legal notes
=================
| SPDX-FileCopyrightText: © 2022 ekvip automation GmbH <info@ekvip.de>
| SPDX-License-Identifier: Apache-2.0
| For details check: Apache-2.0_

.. _Apache-2.0: https://www.apache.org/licenses/LICENSE-2.0

.. </legal notes>

parameters
=================

*)

METHOD win1252IsEqualTo
VAR_INPUT
	(* current string to check *)
	stringToCheck	:POINTER TO BYTE;
	(* ``stringToCheck`` must be equal to expected *)
	expected		:POINTER TO BYTE;
	(* ``TRUE`` means ignore cases; ``FALSE`` means cases must be equal too *)
	ignoreCases		:BOOL;
	(* message if the assertion is false *)
	message			:AssertMessage;
END_VAR
VAR
	(* length of current string to check *)
	lenghtStringToCheck		:UDINT;
	(* length of ``expected`` *)
	lengthExpectedString	:UDINT;
	(* string address we use to compare, if it's case sensitive it's equal to ``stringToCheck`` *)
	usedStringToCheck		:POINTER TO BYTE;
	(* seacrch string address we use to compare, if it's case sensitive it's equal to ``expected`` *)
	usedExpectedString		:POINTER TO BYTE;
END_VAR
VAR CONSTANT
	(* length of an empty string to avoid Tc2_System.MEMCMP with length 0 *)
	EMPTY_STRING_LENGTH		:UDINT := 0;
END_VAR
lenghtStringToCheck := THIS^.getWin1252StringLength(stringToCheck);
lengthExpectedString := THIS^.getWin1252StringLength(expected);

IF (lenghtStringToCheck <> lengthExpectedString) THEN
	THIS^.assertionWasWrong(message, THIS^.getDebugInfo('win1252IsEqualTo'));
	RETURN;
ELSIF (lengthExpectedString = EMPTY_STRING_LENGTH) THEN
	RETURN;
END_IF

usedStringToCheck := THIS^.getNewWin1252UpperCaseString(stringToCheck, lenghtStringToCheck, ignoreCases);
usedExpectedString := THIS^.getNewWin1252UpperCaseString(expected, lengthExpectedString, ignoreCases);

IF (Tc2_System.MEMCMP(
		usedStringToCheck,
		usedExpectedString, 
		lengthExpectedString
	) <> CNM_ReturnTypes.ComparationResult.EQUAL
) THEN
	THIS^.assertionWasWrong(message, THIS^.getDebugInfo('win1252IsEqualTo'));
END_IF;

THIS^.win1252FreeMemory(usedStringToCheck, ignoreCases);
THIS^.win1252FreeMemory(usedExpectedString, ignoreCases);
END_METHOD

(*

short summary
=================
This assertion method for windows-1252 strings checks if the current string ``stringToCheck`` is not equal to the ``unexpected`` string

.. attention:: 
	All strings are handled as null terminated byte streams.
	For windows-1252 is end of the string 16#00

.. <legal notes>

legal notes
=================
| SPDX-FileCopyrightText: © 2022 ekvip automation GmbH <info@ekvip.de>
| SPDX-License-Identifier: Apache-2.0
| For details check: Apache-2.0_

.. _Apache-2.0: https://www.apache.org/licenses/LICENSE-2.0

.. </legal notes>

parameters
=================

*)

METHOD win1252IsNotEqualTo
VAR_INPUT
	(* current string to check *)
	stringToCheck	:POINTER TO BYTE;
	(* ``stringToCheck`` must be not equal to expected *)
	unexpected		:POINTER TO BYTE;
	(* ``TRUE`` means ignore cases; ``FALSE`` means cases must be equal too *)
	ignoreCases		:BOOL;
	(* message if the assertion is false *)
	message			:AssertMessage;
END_VAR
VAR
	(* length of current string to check *)
	lenghtStringToCheck		:UDINT;
	(* length of ``unexpected`` *)
	lengthUnexpectedString	:UDINT;
	(* string address we use to compare, if it's case sensitive it's equal to ``stringToCheck`` *)
	usedStringToCheck		:POINTER TO BYTE;
	(* seacrch string address we use to compare, if it's case sensitive it's equal to ``expected`` *)
	usedUnexpectedString	:POINTER TO BYTE;
END_VAR
VAR CONSTANT
	(* length of an empty string to avoid Tc2_System.MEMCMP with length 0 *)
	EMPTY_STRING_LENGTH		:UDINT := 0;
END_VAR
lenghtStringToCheck := THIS^.getWin1252StringLength(stringToCheck);
lengthUnexpectedString := THIS^.getWin1252StringLength(unexpected);

IF ((lenghtStringToCheck = EMPTY_STRING_LENGTH) AND (lengthUnexpectedString = EMPTY_STRING_LENGTH)) THEN
	THIS^.assertionWasWrong(message, THIS^.getDebugInfo('win1252IsNotEqualTo'));
	RETURN;
END_IF

usedStringToCheck := THIS^.getNewWin1252UpperCaseString(stringToCheck, lenghtStringToCheck, ignoreCases);
usedUnexpectedString := THIS^.getNewWin1252UpperCaseString(unexpected, lengthUnexpectedString, ignoreCases);

IF (Tc2_System.MEMCMP(
		usedStringToCheck,
		usedUnexpectedString, 
		lengthUnexpectedString
	) = CNM_ReturnTypes.ComparationResult.EQUAL
) THEN
	THIS^.assertionWasWrong(message, THIS^.getDebugInfo('win1252IsNotEqualTo'));
END_IF;

THIS^.win1252FreeMemory(usedStringToCheck, ignoreCases);
THIS^.win1252FreeMemory(usedUnexpectedString, ignoreCases);
END_METHOD

(*

short summary
=================
This assertion method checks if the current string ``stringToCheck`` is length
is equal to ``expectedLength``

.. attention:: 
	All strings are handled as null terminated byte streams.
	For windows-1252 is end of the string 16#00

.. <legal notes>

legal notes
=================
| SPDX-FileCopyrightText: © 2022 ekvip automation GmbH <info@ekvip.de>
| SPDX-License-Identifier: Apache-2.0
| For details check: Apache-2.0_

.. _Apache-2.0: https://www.apache.org/licenses/LICENSE-2.0

.. </legal notes>

parameters
=================

*)

METHOD win1252LenghtIsExact
VAR_INPUT
	(* current string to check *)
	stringToCheck	:POINTER TO BYTE;
	(* expected length of ``stringToCheck`` *)
	expectedLength	:UDINT;
	(* message if the assertion is false *)
	message			:AssertMessage;
END_VAR
IF (THIS^.getWin1252StringLength(stringToCheck) <> expectedLength) THEN
	THIS^.assertionWasWrong(message, THIS^.getDebugInfo('win1252LenghtIsExact'));
END_IF
END_METHOD

(*

short summary
=================
This assertion method checks if the current string ``stringToCheck`` is length
is equal or less than to ``maxLength``

.. attention:: 
	All strings are handled as null terminated byte streams.
	For windows-1252 is end of the string 16#00

.. <legal notes>

legal notes
=================
| SPDX-FileCopyrightText: © 2022 ekvip automation GmbH <info@ekvip.de>
| SPDX-License-Identifier: Apache-2.0
| For details check: Apache-2.0_

.. _Apache-2.0: https://www.apache.org/licenses/LICENSE-2.0

.. </legal notes>

parameters
=================

*)

METHOD win1252LenghtIsMax
VAR_INPUT
	(* current string to check *)
	stringToCheck	:POINTER TO BYTE;
	(* upper limit of the length of ``stringToCheck`` *)
	maxLength		:UDINT;
	(* message if the assertion is false *)
	message			:AssertMessage;
END_VAR
IF (THIS^.getWin1252StringLength(stringToCheck) > maxLength) THEN
	THIS^.assertionWasWrong(message, THIS^.getDebugInfo('win1252LenghtIsMax'));
END_IF
END_METHOD

(*

short summary
=================
This assertion method checks if the current string ``stringToCheck`` is length
is equal or grater than to ``minLength``

.. attention:: 
	All strings are handled as null terminated byte streams.
	For windows-1252 is end of the string 16#00

.. <legal notes>

legal notes
=================
| SPDX-FileCopyrightText: © 2022 ekvip automation GmbH <info@ekvip.de>
| SPDX-License-Identifier: Apache-2.0
| For details check: Apache-2.0_

.. _Apache-2.0: https://www.apache.org/licenses/LICENSE-2.0

.. </legal notes>

parameters
=================

*)

METHOD win1252LenghtIsMin
VAR_INPUT
	(* current string to check *)
	stringToCheck	:POINTER TO BYTE;
	(* lower limit of the length of ``stringToCheck`` *)
	minLength		:UDINT;
	(* message if the assertion is false *)
	message			:AssertMessage;
END_VAR
IF (THIS^.getWin1252StringLength(stringToCheck) < minLength) THEN
	THIS^.assertionWasWrong(message, THIS^.getDebugInfo('win1252LenghtIsMin'));
END_IF
END_METHOD

(*

short summary
=================
This assertion method checks if the current string ``stringToCheck`` is length
is equal or grater than ``minLength`` and equal or less than ``maxLength``

.. attention:: 
	All strings are handled as null terminated byte streams.
	For windows-1252 is end of the string 16#00

.. <legal notes>

legal notes
=================
| SPDX-FileCopyrightText: © 2022 ekvip automation GmbH <info@ekvip.de>
| SPDX-License-Identifier: Apache-2.0
| For details check: Apache-2.0_

.. _Apache-2.0: https://www.apache.org/licenses/LICENSE-2.0

.. </legal notes>

parameters
=================

*)

METHOD win1252LengthIsBetween
VAR_INPUT
	(* current string to check *)
	stringToCheck	:POINTER TO BYTE;
	(* lower limit of the string length *)
	minLenght		:UDINT;
	(* upper limit of the string length *)
	maxLenght		:UDINT;
	(* message if the assertion is false *)
	message			:AssertMessage;
END_VAR
VAR
	(* length of ``stringToCheck`` *)
	lenghtStringToCheck	:UDINT;
END_VAR
IF (minLenght > maxLenght) THEN
	THIS^.assertionWasWrong(message, THIS^.getDebugInfo('win1252LengthIsBetween'));
	RETURN;
END_IF

lenghtStringToCheck := THIS^.getWin1252StringLength(stringToCheck);

IF (
	(lenghtStringToCheck < minLenght)
	OR (lenghtStringToCheck > maxLenght)
) THEN
	THIS^.assertionWasWrong(message, THIS^.getDebugInfo('win1252LengthIsBetween'));
END_IF;
END_METHOD

(*

short summary
=================
This assertion method checks if the current string ``stringToCheck`` starts with ``start``

.. attention:: 
	All strings are handled as null terminated byte streams.
	For windows-1252 is end of the string 16#00

.. <legal notes>

legal notes
=================
| SPDX-FileCopyrightText: © 2022 ekvip automation GmbH <info@ekvip.de>
| SPDX-License-Identifier: Apache-2.0
| For details check: Apache-2.0_

.. _Apache-2.0: https://www.apache.org/licenses/LICENSE-2.0

.. </legal notes>

parameters
=================

*)

METHOD win1252StartsWith
VAR_INPUT
	(* current string to check *)
	stringToCheck	:POINTER TO BYTE;
	(* expected start of ``stringToCheck`` *)
	start			:POINTER TO BYTE;
	(* ``TRUE`` means ignore cases; ``FALSE`` means cases must be equal too *)
	ignoreCases		:BOOL;
	(* ``TRUE`` means truncation of spaces on the left side of ``stringToCheck``*)
	trim			:BOOL;
	(* message if the assertion is false *)
	message			:AssertMessage;
END_VAR
VAR
	(* length of current string to check *)
	lenghtStringToCheck	:UDINT;
	(* length of ``start`` *)
	lengthOfStart		:UDINT;
	(* string address we use to compare, if it's case sensitive it's equal to ``stringToCheck`` *)
	usedStringToCheck	:POINTER TO BYTE;
	(* seacrch string address we use to compare, if it's case sensitive it's equal to ``start`` *)
	usedStartString		:POINTER TO BYTE;
END_VAR
lenghtStringToCheck := THIS^.getWin1252StringLength(stringToCheck);
lengthOfStart := THIS^.getWin1252StringLength(start);

THIS^.win1252TrimLeft(stringToCheck, lenghtStringToCheck, trim);

IF (
	NOT THIS^.isContainsCheckNecessary(
		stringToCheck		:= stringToCheck,
		searchString		:= start,
		lenghtStringToCheck	:= lenghtStringToCheck,
		lengthSearchString	:= lengthOfStart,
		additionalText		:= THIS^.getDebugInfo('win1252StartsWith'),
		message				:= message
	)
) THEN
	RETURN;
END_IF

usedStringToCheck := THIS^.getNewWin1252UpperCaseString(stringToCheck, lenghtStringToCheck, ignoreCases);
usedStartString := THIS^.getNewWin1252UpperCaseString(start, lengthOfStart, ignoreCases);

IF (Tc2_System.MEMCMP(
		usedStringToCheck,
		usedStartString, 
		lengthOfStart
	) <> CNM_ReturnTypes.ComparationResult.EQUAL
) THEN
	THIS^.assertionWasWrong(message, THIS^.getDebugInfo('win1252StartsWith'));
END_IF;

THIS^.win1252FreeMemory(usedStringToCheck, ignoreCases);
THIS^.win1252FreeMemory(usedStartString, ignoreCases);
END_METHOD

(*

short summary
=================
This method is used to remove the whitespace from the start of the string.
It does not really remove it, it just moves the start address and decreases
the string length

.. <legal notes>

legal notes
=================
| SPDX-FileCopyrightText: © 2022 ekvip automation GmbH <info@ekvip.de>
| SPDX-License-Identifier: Apache-2.0
| For details check: Apache-2.0_

.. _Apache-2.0: https://www.apache.org/licenses/LICENSE-2.0

.. </legal notes>

parameters
=================

*)

METHOD PROTECTED win1252TrimLeft
VAR_IN_OUT
	(* start address of the string *)
	stringAddress	:POINTER TO BYTE;
	(* length of the string ``stringAddress`` *)
	stringLength	:UDINT;
END_VAR
VAR_INPUT
	(* ``TRUE`` means remove the whitespace, ``FALSE`` means do not remove the whitespace *)
	trimString		:BOOL;
END_VAR
VAR
	(* index of the current character *)
	character		:UDINT;
	(* counter of the whitspace characters *)
	whitespaceCount	:UDINT := 0;
END_VAR
IF ((stringAddress = 0) OR (stringLength <= 0) OR (NOT trimString)) THEN
	RETURN;
END_IF

FOR character := 0 TO (stringLength-1) BY 1 DO
	IF (THIS^.isCharWin1252WhiteSpace(stringAddress[character])) THEN
		whitespaceCount := whitespaceCount + 1;
	ELSE
		EXIT;
	END_IF
END_FOR

stringAddress := ADR(stringAddress[whitespaceCount]);
stringLength := stringLength - whitespaceCount;
END_METHOD

(*

short summary
=================
This method is used to remove the whitespace from the end of the string.
It does not really remove it, it just decreases the string length.

.. <legal notes>

legal notes
=================
| SPDX-FileCopyrightText: © 2022 ekvip automation GmbH <info@ekvip.de>
| SPDX-License-Identifier: Apache-2.0
| For details check: Apache-2.0_

.. _Apache-2.0: https://www.apache.org/licenses/LICENSE-2.0

.. </legal notes>

parameters
=================

*)

METHOD PROTECTED win1252TrimRight
VAR_INPUT
	(* start address of the string *)
	stringAddress	:POINTER TO BYTE;
END_VAR
VAR_IN_OUT
	(* length of the string ``stringAddress`` *)
	stringLength	:UDINT;
END_VAR
VAR_INPUT
	(* ``TRUE`` means remove the whitespace, ``FALSE`` means do not remove the whitespace *)
	trimString		:BOOL;
END_VAR
VAR
	(* index of the current character *)
	character	:LINT;
END_VAR
IF ((stringAddress = 0) OR (stringLength <= 0) OR (NOT trimString)) THEN
	RETURN;
END_IF

FOR character := (stringLength-1) TO 0 BY -1 DO
	IF (THIS^.isCharWin1252WhiteSpace(stringAddress[character])) THEN
		stringLength := stringLength-1;
	ELSE
		RETURN;
	END_IF
END_FOR
END_METHOD

(*

short summary
=================
This method converts the lowercase letters in an 8 bit windows-1252 string to uppercase letters.

.. attention:: 
	All strings are handled as null terminated byte streams.
	For windows-1252 is end of the string 16#00

.. attention::
	Sharp S ß (16#DF) will not converted

.. <legal notes>

legal notes
=================
| SPDX-FileCopyrightText: © 2022 ekvip automation GmbH <info@ekvip.de>
| SPDX-License-Identifier: Apache-2.0
| For details check: Apache-2.0_

.. _Apache-2.0: https://www.apache.org/licenses/LICENSE-2.0

.. </legal notes>

parameters
=================

*)

METHOD PROTECTED win1252UpperCase
VAR_INPUT
	(* string to ucase *)
	stringAddress		:POINTER TO BYTE;
	(* length of the string *)
	stringLength		:UDINT;
END_VAR
VAR
	(* index of the current character *)
	character			:UDINT := 0;
END_VAR
VAR CONSTANT
	(* NUL: $00 *)
	END_OF_STRING							:BYTE := 16#00;
	(* a *)                             	
	LOWERCASE_A								:BYTE := 16#61;
	(* z *)                             	
	LOWERCASE_Z								:BYTE := 16#7A;
	(* ß *)                             	
	LOWERCASE_SHARP_S						:BYTE := 16#DF;
	(* ÿ *)                             	
	LOWERCASE_Y_WITH_DIAERESIS				:BYTE := 16#FF;
	(* Ÿ *)                             	
	UPPERCASE_Y_WITH_DIAERESIS				:BYTE := 16#9F;
	(* à *)                             	
	LOWERCASE_A_WITH_GRAVE					:BYTE := 16#E0;
	(* ö *)                             	
	LOWERCASE_O_WITH_DIAERESIS				:BYTE := 16#F6;
	(* ø *)                             	
	LOWERCASE_O_WITH_SLASH					:BYTE := 16#F8;
	(* þ *)                             	
	LOWERCASE_THORN							:BYTE := 16#FE;
	(* š *)                             	
	LOWERCASE_S_WITH_CARON					:BYTE := 16#9A;
	(* œ *)                             	
	LOWERCASE_OE							:BYTE := 16#9C;
	(* ž *)                             	
	LOWERCASE_Z_WITH_CARON					:BYTE := 16#9E;
	(* difference between lowercase and uppercase except for š,œ and ž *)
	DIFFERENCE_LOWERCASE_UPPERCASE			:BYTE := 16#20;
	(* for š,œ and ž the difference between lowercase and uppercase *)
	DIFFERENCE_LOWERCASE_UPPERCASE_SPECIAL	:BYTE := 16#10;
	(* increment for the character index *)
	INCREMENT_CHARACTER						:UDINT := 1;
END_VAR
IF (stringAddress = 0) THEN
	RETURN;
END_IF

WHILE ((stringAddress[character] <> END_OF_STRING) AND (character <= stringLength)) DO
	CASE stringAddress[character] OF
	LOWERCASE_A..LOWERCASE_Z,
	LOWERCASE_A_WITH_GRAVE..LOWERCASE_O_WITH_DIAERESIS,
	LOWERCASE_O_WITH_SLASH..LOWERCASE_THORN:
		stringAddress[character] := stringAddress[character] - DIFFERENCE_LOWERCASE_UPPERCASE;
	LOWERCASE_S_WITH_CARON,
	LOWERCASE_OE,
	LOWERCASE_Z_WITH_CARON:
		stringAddress[character] := stringAddress[character] - DIFFERENCE_LOWERCASE_UPPERCASE_SPECIAL;
	LOWERCASE_Y_WITH_DIAERESIS:
		stringAddress[character] := UPPERCASE_Y_WITH_DIAERESIS;
	LOWERCASE_SHARP_S:;//for ß do nothing, because there is no capital letter for it
	ELSE;// do nothing, it's no small letter 
	END_CASE
	character := character + INCREMENT_CHARACTER;
END_WHILE
END_METHOD

END_FUNCTION_BLOCK

// ---- Assertor/Assertions/StringAssertion/classes/AbstarctStringPointerAssertions.TcPOU
(*

short summary
=================
Abstract class provides methods for checking whether, 
based on the string lengths an assert statement with contains or contains not,
makes sense

.. <legal notes>

legal notes
=================
| SPDX-FileCopyrightText: © 2022 ekvip automation GmbH <info@ekvip.de>
| SPDX-License-Identifier: Apache-2.0
| For details check: Apache-2.0_

.. _Apache-2.0: https://www.apache.org/licenses/LICENSE-2.0

.. </legal notes>

methods and properties
=======================

*)

{attribute 'reflection'}
FUNCTION_BLOCK INTERNAL ABSTRACT AbstarctStringPointerAssertions EXTENDS AbstactAssertion 
VAR
END_VAR

(*

short summary
=================
This abstract property returns the class name of the concrete object, 
It's for debugging purpose

.. attention:: 
	For derivations: **It is necessary that this property is overridden by the concrete class**

.. <legal notes>

legal notes
=================
| SPDX-FileCopyrightText: © 2022 ekvip automation GmbH <info@ekvip.de>
| SPDX-License-Identifier: Apache-2.0
| For details check: Apache-2.0_

.. _Apache-2.0: https://www.apache.org/licenses/LICENSE-2.0

.. </legal notes>

*)

PROPERTY ABSTRACT className :CNM_AbstractObject.ClassName
GET
END_GET
END_PROPERTY

(*

short summary
=================
Methods for checking whether, based on the string lengths an assert statement with contains makes sense

.. <legal notes>

legal notes
=================
| SPDX-FileCopyrightText: © 2022 ekvip automation GmbH <info@ekvip.de>
| SPDX-License-Identifier: Apache-2.0
| For details check: Apache-2.0_

.. _Apache-2.0: https://www.apache.org/licenses/LICENSE-2.0

.. </legal notes>

parameters
==================
:return: ``FLASE`` means it's not necessary 
to check the string content, ``TRUE`` means
it's necessary to check the string content
to know if the assertion is true or false

*)

METHOD PROTECTED isContainsCheckNecessary :BOOL
VAR_INPUT
	(* current string to check *)
	stringToCheck	:POINTER TO BYTE;
	(* string must be found in ``stringToCheck`` *)
	searchString		:POINTER TO BYTE;
	(* length of current string to check *)
	lenghtStringToCheck	:UDINT;
	(* length of ``searchString`` *)
	lengthSearchString	:UDINT;
	(* just additional text if assert is false *)	
	additionalText		:Tc2_System.T_MaxString;
	(* message if the assertion is false *)
	message				:AssertMessage;
END_VAR
isContainsCheckNecessary := FALSE;
IF (lengthSearchString > lenghtStringToCheck) THEN
	THIS^.assertionWasWrong(message, additionalText);
	RETURN;
ELSIF ((stringToCheck = 0) XOR (searchString = 0)) THEN
	THIS^.assertionWasWrong(message, additionalText);
	RETURN;
ELSIF ((stringToCheck = 0) AND (searchString = 0)) THEN
	RETURN; //assert is true
ELSIF (lengthSearchString = 0) THEN
	RETURN; //assert is true
ELSIF ((lenghtStringToCheck <= 0) AND (lengthSearchString > 0)) THEN
	THIS^.assertionWasWrong(message, additionalText);
	RETURN;
END_IF
isContainsCheckNecessary := TRUE;
END_METHOD

(*

short summary
=================
Methods for checking whether, based on the string lengths an assert statement with containsNo makes sense

.. <legal notes>

legal notes
=================
| SPDX-FileCopyrightText: © 2022 ekvip automation GmbH <info@ekvip.de>
| SPDX-License-Identifier: Apache-2.0
| For details check: Apache-2.0_

.. _Apache-2.0: https://www.apache.org/licenses/LICENSE-2.0

.. </legal notes>

parameters
==================
:return: ``FLASE`` means it's not necessary 
to check the string content, ``TRUE`` means
it's necessary to check the string content
to know if the assertion is true or false

*)

METHOD PROTECTED isContainsNoCheckNecessary :BOOL
VAR_INPUT
	(* current string to check *)
	stringToCheck		:POINTER TO BYTE;
	(* string must be found in ``stringToCheck`` *)
	searchString		:POINTER TO BYTE;
	(* length of current string to check *)
	lenghtStringToCheck	:UDINT;
	(* length of ``searchString`` *)
	lengthSearchString	:UDINT;
	(* just additional text if assert is false *)	
	additionalText		:Tc2_System.T_MaxString;
	(* message if the assertion is false *)
	message				:AssertMessage;
END_VAR
isContainsNoCheckNecessary := FALSE;
IF (lengthSearchString > lenghtStringToCheck) THEN
	RETURN; //assert is true
ELSIF ((stringToCheck = 0) XOR (searchString = 0)) THEN
	RETURN; //assert is true
ELSIF ((stringToCheck = 0) AND (searchString = 0)) THEN
	THIS^.assertionWasWrong(message, additionalText);
	RETURN;
ELSIF (lengthSearchString = 0) THEN
	THIS^.assertionWasWrong(message, additionalText);
	RETURN;
ELSIF ((lenghtStringToCheck <= 0) AND (lengthSearchString > 0)) THEN
	RETURN; //assert is true
END_IF
isContainsNoCheckNecessary := TRUE;
END_METHOD

END_FUNCTION_BLOCK

// ---- Assertor/Assertions/StringAssertion/StringNew/classes/Windows125xStringAssertions.TcPOU
(*

short summary
=================
This class provides assert statements for Windows-1252 and Windows-1251 strings up to 255 characters length. 
Used encoding is specified in ``Tc2_Utilities.GLOBAL_SBCS_TABLE`` global variable

.. attention:: 
	All strings are handled as null-terminated byte streams

.. <legal notes>

legal notes
=================
| SPDX-FileCopyrightText: © 2024 ekvip automation GmbH <info@ekvip.de>
| SPDX-License-Identifier: Apache-2.0
| For details check: Apache-2.0_

.. _Apache-2.0: https://www.apache.org/licenses/LICENSE-2.0

.. </legal notes>

methods and properties
=======================

*)

{attribute 'reflection'}
FUNCTION_BLOCK INTERNAL Windows125xStringAssertions EXTENDS AbstactAssertion IMPLEMENTS IWindows125xStringAssertions
VAR
	(* class to handle the windows-1252 and windows-1251 string assertions *)  
	assertion	:Windows125xStringPointerAssertions();
END_VAR

(*

short summary
=================
This abstract property returns the class name of the concrete object, 
It's for debugging purpose

.. <legal notes>

legal notes
=================
| SPDX-FileCopyrightText: © 2022 ekvip automation GmbH <info@ekvip.de>
| SPDX-License-Identifier: Apache-2.0
| For details check: Apache-2.0_

.. _Apache-2.0: https://www.apache.org/licenses/LICENSE-2.0

.. </legal notes>

*)

PROPERTY className :CNM_AbstractObject.ClassName
GET
className := 'CNM_AssertionInterfaceLib.Windows125xStringAssertions';
END_GET
END_PROPERTY

(*

short summary
=================
This assertion method checks if the current string ``stringToCheck`` contains the search string ``searchString``.
Processed strings must be in UTF-8 encoding

.. <legal notes>

legal notes
=================
| SPDX-FileCopyrightText: © 2024 ekvip automation GmbH <info@ekvip.de>
| SPDX-License-Identifier: Apache-2.0
| For details check: Apache-2.0_

.. _Apache-2.0: https://www.apache.org/licenses/LICENSE-2.0

.. </legal notes>

parameters
=================

*)

METHOD contains : IWindows125xStringAssertions
VAR_INPUT
	(* current string to check *)
	stringToCheck	:Tc2_System.T_MaxString;
	(* string must be found in ``stringToCheck`` *)
	searchString	:Tc2_System.T_MaxString;
	(* ``TRUE`` means ignore cases; ``FALSE`` means that cases must be equal too *)
	ignoreCases		:BOOL;
	(* message if the assertion is false *)
	message			:AssertMessage;
END_VAR
contains := THIS^;

assertion.contains(
	stringToCheck 	:= ADR(stringToCheck),
	searchSTring 	:= ADR(searchString),
	ignoreCases 	:= ignoreCases,
	message 		:= message
);
END_METHOD

(*

short summary
=================
This assertion method checks if the current string ``stringToCheck`` doesn't contain the search string ``searchString``.
Processed strings must be in UTF-8 encoding

.. <legal notes>

legal notes
=================
| SPDX-FileCopyrightText: © 2024 ekvip automation GmbH <info@ekvip.de>
| SPDX-License-Identifier: Apache-2.0
| For details check: Apache-2.0_

.. _Apache-2.0: https://www.apache.org/licenses/LICENSE-2.0

.. </legal notes>

parameters
=================

*)

METHOD containsNo : IWindows125xStringAssertions
VAR_INPUT
	(* current string to check *)
	stringToCheck	:Tc2_System.T_MaxString;
	(* string that must not be found in ``stringToCheck`` *)
	searchString	:Tc2_System.T_MaxString;
	(* ``TRUE`` means ignore cases; ``FALSE`` means that cases must be equal too *)
	ignoreCases		:BOOL;
	(* message if the assertion is false *)
	message			:AssertMessage;
END_VAR
containsNo := THIS^;

THIS^.assertion.containsNo(
	stringToCheck 	:= ADR(stringToCheck),
	searchSTring 	:= ADR(searchString),
	ignoreCases 	:= ignoreCases,
	message 		:= message
);
END_METHOD

(*

short summary
=================
This assertion method checks if the current string ``stringToCheck`` ends with the string ``end``.
Processed strings must be in UTF-8 encoding

.. <legal notes>

legal notes
=================
| SPDX-FileCopyrightText: © 2024 ekvip automation GmbH <info@ekvip.de>
| SPDX-License-Identifier: Apache-2.0
| For details check: Apache-2.0_

.. _Apache-2.0: https://www.apache.org/licenses/LICENSE-2.0

.. </legal notes>

parameters
=================

*)

METHOD endsWith : IWindows125xStringAssertions
VAR_INPUT
	(* current string to check *)
	stringToCheck	:Tc2_System.T_MaxString;
	(* expected end of ``stringToCheck`` *)
	end				:Tc2_System.T_MaxString;
	(* ``TRUE`` means ignore cases; ``FALSE`` means that cases must be equal too *)
	ignoreCases		:BOOL;
	(* ``TRUE`` means truncation of spaces on the right side of ``stringToCheck``*)
	trimRight		:BOOL;
	(* message if the assertion is false *)
	message			:AssertMessage;
END_VAR
endsWith := THIS^;

assertion.endsWith(
	stringToCheck	:= ADR(stringToCheck),
	end				:= ADR(end),
	ignoreCases		:= ignoreCases,
	trimRight		:= trimRight,
	message			:= message
);
END_METHOD

(*

short summary
=================
This assertion method checks if the current string ``stringToCheck`` is empty.
Processed strings must be in UTF-8 encoding

.. <legal notes>

legal notes
=================
| SPDX-FileCopyrightText: © 2024 ekvip automation GmbH <info@ekvip.de>
| SPDX-License-Identifier: Apache-2.0
| For details check: Apache-2.0_

.. _Apache-2.0: https://www.apache.org/licenses/LICENSE-2.0

.. </legal notes>

parameters
=================

*)

METHOD isEmpty : IWindows125xStringAssertions
VAR_INPUT
	(* current string to check *)
	stringToCheck	:Tc2_System.T_MaxString;
	(* message if the assertion is false *)
	message			:AssertMessage;
END_VAR
isEmpty := THIS^;

IF (stringToCheck <> '') THEN
	THIS^.assertionWasWrong(message, THIS^.getDebugInfo('isEmpty'));
END_IF
END_METHOD

(*

short summary
=================
This assertion method checks if the current string ``stringToCheck`` is equal to ``expected``.
Processed strings must be in UTF-8 encoding

.. <legal notes>

legal notes
=================
| SPDX-FileCopyrightText: © 2024 ekvip automation GmbH <info@ekvip.de>
| SPDX-License-Identifier: Apache-2.0
| For details check: Apache-2.0_

.. _Apache-2.0: https://www.apache.org/licenses/LICENSE-2.0

.. </legal notes>

parameters
=================

*)

METHOD isEqualTo : IWindows125xStringAssertions
VAR_INPUT
	(* current string to check *)
	stringToCheck	:Tc2_System.T_MaxString;
	(* ``stringToCheck`` must be equal to expected *)
	expected		:Tc2_System.T_MaxString;
	(* ``TRUE`` means ignore cases; ``FALSE`` means that cases must be equal too *)
	ignoreCases		:BOOL;
	(* message if the assertion is false *)
	message			:AssertMessage;
END_VAR
isEqualTo := THIS^;

assertion.isEqualTo(
	stringToCheck	:= ADR(stringToCheck),
	expected		:= ADR(expected),
	ignoreCases		:= ignoreCases,
	message			:= message
);
END_METHOD

(*

short summary
=================
This assertion method checks if the current string ``stringToCheck`` is not empty.
Processed strings must be in UTF-8 encoding

.. <legal notes>

legal notes
=================
| SPDX-FileCopyrightText: © 2024 ekvip automation GmbH <info@ekvip.de>
| SPDX-License-Identifier: Apache-2.0
| For details check: Apache-2.0_

.. _Apache-2.0: https://www.apache.org/licenses/LICENSE-2.0

.. </legal notes>

parameters
=================

*)

METHOD isNotEmpty : IWindows125xStringAssertions
VAR_INPUT
	(* current string to check *)
	stringToCheck	:Tc2_System.T_MaxString;
	(* message if the assertion is false *)
	message			:AssertMessage;
END_VAR
isNotEmpty := THIS^;

IF (stringToCheck = '') THEN
	THIS^.assertionWasWrong(message, THIS^.getDebugInfo('isEmpty'));
END_IF
END_METHOD

(*

short summary
=================
This assertion method checks if the current string ``stringToCheck`` is not equal to ``unexpected``.
Processed strings must be in UTF-8 encoding

.. <legal notes>

legal notes
=================
| SPDX-FileCopyrightText: © 2024 ekvip automation GmbH <info@ekvip.de>
| SPDX-License-Identifier: Apache-2.0
| For details check: Apache-2.0_

.. _Apache-2.0: https://www.apache.org/licenses/LICENSE-2.0

.. </legal notes>

parameters
=================

*)

METHOD isNotEqualTo : IWindows125xStringAssertions
VAR_INPUT
	(* current string to check *)
	stringToCheck	:Tc2_System.T_MaxString;
	(* ``stringToCheck`` must be not equal to expected *)
	unexpected		:Tc2_System.T_MaxString;
	(* ``TRUE`` means ignore cases; ``FALSE`` means that cases must be equal too *)
	ignoreCases		:BOOL;
	(* message if the assertion is false *)
	message			:AssertMessage;
END_VAR
isNotEqualTo := THIS^;

THIS^.assertion.isNotEqualTo(
	stringToCheck	:= ADR(stringToCheck),
	unexpected		:= ADR(unexpected),
	ignoreCases		:= ignoreCases,
	message			:= message
);
END_METHOD

(*

short summary
=================
This assertion method checks if the current string ``stringToCheck`` length is between ``minLenght`` and ``maxLenght``.
Processed strings must be in UTF-8 encoding

.. <legal notes>

legal notes
=================
| SPDX-FileCopyrightText: © 2024 ekvip automation GmbH <info@ekvip.de>
| SPDX-License-Identifier: Apache-2.0
| For details check: Apache-2.0_

.. _Apache-2.0: https://www.apache.org/licenses/LICENSE-2.0

.. </legal notes>

parameters
=================

*)

METHOD lenghtIsBetween : IWindows125xStringAssertions
VAR_INPUT
	(* current string to check *)
	stringToCheck	:Tc2_System.T_MaxString;
	(* lower limit of the string length *)
	minLenght		:USINT;
	(* upper limit of the string length *)
	maxLenght		:USINT;
	(* message if the assertion is false *)
	message			:AssertMessage;
END_VAR
lenghtIsBetween := THIS^;

THIS^.assertion.lengthIsBetween(
	stringToCheck	:= ADR(stringToCheck),
	minLenght		:= minLenght,
	maxLenght		:= maxLenght,
	message			:= message
);
END_METHOD

(*

short summary
=================
This assertion method checks if the current string ``stringToCheck`` length is equal to ``expectedLength``.
Processed strings must be in UTF-8 encoding

.. <legal notes>

legal notes
=================
| SPDX-FileCopyrightText: © 2024 ekvip automation GmbH <info@ekvip.de>
| SPDX-License-Identifier: Apache-2.0
| For details check: Apache-2.0_

.. _Apache-2.0: https://www.apache.org/licenses/LICENSE-2.0

.. </legal notes>

parameters
=================

*)

METHOD lenghtIsExact : IWindows125xStringAssertions
VAR_INPUT
	(* current string to check *)
	stringToCheck	:Tc2_System.T_MaxString;
	(* expected length of ``stringToCheck`` *)
	expectedLength	:USINT;
	(* message if the assertion is false *)
	message			:AssertMessage;
END_VAR
lenghtIsExact := THIS^;

THIS^.assertion.lenghtIsExact(
	stringToCheck	:= ADR(stringToCheck),
	expectedLength	:= expectedLength,
	message			:= message
);
END_METHOD

(*

short summary
=================
This assertion method checks if the current string ``stringToCheck`` length is equal or less than to ``maxLength``.
Processed strings must be in UTF-8 encoding

.. <legal notes>

legal notes
=================
| SPDX-FileCopyrightText: © 2024 ekvip automation GmbH <info@ekvip.de>
| SPDX-License-Identifier: Apache-2.0
| For details check: Apache-2.0_

.. _Apache-2.0: https://www.apache.org/licenses/LICENSE-2.0

.. </legal notes>

parameters
=================

*)

METHOD lenghtIsMax : IWindows125xStringAssertions
VAR_INPUT
	(* current string to check *)
	stringToCheck	:Tc2_System.T_MaxString;
	(* upper limit of the length of ``stringToCheck`` *)
	maxLength		:USINT;
	(* message if the assertion is false *)
	message			:AssertMessage;
END_VAR
lenghtIsMax := THIS^;

THIS^.assertion.lenghtIsMax(
	stringToCheck	:= ADR(stringToCheck),
	maxLength		:= maxLength,
	message			:= message
);
END_METHOD

(*

short summary
=================
This assertion method checks if the current string ``stringToCheck`` length is equal or grater than to ``minLength``.
Processed strings must be in UTF-8 encoding

.. <legal notes>

legal notes
=================
| SPDX-FileCopyrightText: © 2024 ekvip automation GmbH <info@ekvip.de>
| SPDX-License-Identifier: Apache-2.0
| For details check: Apache-2.0_

.. _Apache-2.0: https://www.apache.org/licenses/LICENSE-2.0

.. </legal notes>

parameters
=================

*)

METHOD lenghtIsMin : IWindows125xStringAssertions
VAR_INPUT
	(* current string to check *)
	stringToCheck	:Tc2_System.T_MaxString;
	(* lower limit of the length of ``stringToCheck`` *)
	minLength		:USINT;
	(* message if the assertion is false *)
	message			:AssertMessage;
END_VAR
lenghtIsMin := THIS^;

THIS^.assertion.lenghtIsMin(
	stringToCheck	:= ADR(stringToCheck),
	minLength		:= minLength,
	message			:= message
);
END_METHOD

(*

short summary
=================
This methods is the setter for the callback class if an assertion was false

.. <legal notes>

legal notes
=================
| SPDX-FileCopyrightText: © 2024 ekvip automation GmbH <info@ekvip.de>
| SPDX-License-Identifier: Apache-2.0
| For details check: Apache-2.0_

.. _Apache-2.0: https://www.apache.org/licenses/LICENSE-2.0

.. </legal notes>

parameters
=================

*)

METHOD setCallBack
VAR_INPUT
	(* the class that must be informed if an assertion is false *)
	callBack	:IAssertCallback;  
END_VAR
SUPER^.setCallBack(callBack);
THIS^.assertion.setCallBack(callBack);
END_METHOD

(*

short summary
=================
This assertion method checks if the current string ``stringToCheck`` starts with string ``start``.
Processed strings must be in UTF-8 encoding

.. <legal notes>

legal notes
=================
| SPDX-FileCopyrightText: © 2024 ekvip automation GmbH <info@ekvip.de>
| SPDX-License-Identifier: Apache-2.0
| For details check: Apache-2.0_

.. _Apache-2.0: https://www.apache.org/licenses/LICENSE-2.0

.. </legal notes>

parameters
=================

*)

METHOD startsWith : IWindows125xStringAssertions
VAR_INPUT
	(* current string to check *)
	stringToCheck	:Tc2_System.T_MaxString;
	(* expected start of ``stringToCheck`` *)
	start			:Tc2_System.T_MaxString;
	(* ``TRUE`` means ignore cases; ``FALSE`` means that cases must be equal too *)
	ignoreCases		:BOOL;
	(* ``TRUE`` means truncation of spaces on the left side of ``stringToCheck``*)
	trimLeft		:BOOL;
	(* message if the assertion is false *)
	message			:AssertMessage;
END_VAR
startsWith := THIS^;

assertion.startsWith(
	stringToCheck	:= ADR(stringToCheck),
	start			:= ADR(start),
	ignoreCases		:= ignoreCases,
	trimLeft		:= trimLeft,
	message			:= message
);
END_METHOD

END_FUNCTION_BLOCK

// ---- Assertor/Assertions/StringAssertion/StringNew/classes/Windows125xStringPointerAssertions.TcPOU
(*

short summary
=================
This class provides assert statements for Windows-1252 and Windows-1251 strings.
Used encoding is specified in ``Tc2_Utilities.GLOBAL_SBCS_TABLE`` global variable

.. attention:: 
	All strings are handled as null-terminated byte streams

.. <legal notes>

legal notes
=================
| SPDX-FileCopyrightText: © 2024 ekvip automation GmbH <info@ekvip.de>
| SPDX-License-Identifier: Apache-2.0
| For details check: Apache-2.0_

.. _Apache-2.0: https://www.apache.org/licenses/LICENSE-2.0

.. </legal notes>

methods and properties
=======================

*)

{attribute 'reflection'}
FUNCTION_BLOCK INTERNAL Windows125xStringPointerAssertions EXTENDS AbstarctStringPointerAssertions IMPLEMENTS IWindows125xStringPointerAssertions

(*

short summary
=================
This abstract property returns the class name of the concrete object, 
It's for debugging purpose

.. <legal notes>

legal notes
=================
| SPDX-FileCopyrightText: © 2024 ekvip automation GmbH <info@ekvip.de>
| SPDX-License-Identifier: Apache-2.0
| For details check: Apache-2.0_

.. _Apache-2.0: https://www.apache.org/licenses/LICENSE-2.0

.. </legal notes>

*)

PROPERTY className :CNM_AbstractObject.ClassName
GET
className := 'CNM_AssertionInterfaceLib.Windows125xStringPointerAssertions';
END_GET
END_PROPERTY

(*

short summary
=================
This assertion method checks if the current string ``stringToCheck`` contains the search string ``searchString``.
Processed strings must be in Windows-1252 or Windows-1251 encoding

.. attention:: 
	All strings are handled as null-terminated byte streams

.. <legal notes>

legal notes
=================
| SPDX-FileCopyrightText: © 2024 ekvip automation GmbH <info@ekvip.de>
| SPDX-License-Identifier: Apache-2.0
| For details check: Apache-2.0_

.. _Apache-2.0: https://www.apache.org/licenses/LICENSE-2.0

.. </legal notes>

parameters
=================

*)

METHOD contains : IWindows125xStringPointerAssertions
VAR_INPUT
	(* current string to check *)
	stringToCheck	:POINTER TO BYTE;
	(* string must be found in ``stringToCheck`` *)
	searchString	:POINTER TO BYTE;
	(* ``TRUE`` means ignore cases; ``FALSE`` means that cases must be equal too *)
	ignoreCases		:BOOL;
	(* message if the assertion is false *)
	message			:AssertMessage;
END_VAR
VAR
	(* length of current string to check *)
	lenghtStringToCheck	:UDINT;
	(* length of ``searchString`` *)
	lengthSearchString	:UDINT;
	(* string address we use to compare, if it's case sensitive it's equal to ``stringToCheck`` *)
	usedStringToCheck	:POINTER TO BYTE;
	(* seacrch string address we use to compare, if it's case sensitive it's equal to ``searchString`` *)
	usedSearchString	:POINTER TO BYTE;
	(* character index for the comperation *)
	character			:UDINT;
END_VAR
contains := THIS^;

lenghtStringToCheck := THIS^.getStringLength(stringToCheck);
lengthSearchString := THIS^.getStringLength(searchString);

IF (
	NOT THIS^.isContainsCheckNecessary(
		stringToCheck		:= stringToCheck,
		searchString		:= searchString,
		lenghtStringToCheck	:= lenghtStringToCheck,
		lengthSearchString	:= lengthSearchString,
		additionalText		:= THIS^.getDebugInfo('contains'),
		message				:= message
	)
) THEN
	RETURN;
END_IF

usedStringToCheck := THIS^.getNewUpperCaseString(stringToCheck, lenghtStringToCheck, ignoreCases);
usedSearchString := THIS^.getNewUpperCaseString(searchString, lengthSearchString, ignoreCases);

FOR (character := 0) TO (lenghtStringToCheck - lengthSearchString) BY 1 DO
	IF (Tc2_System.MEMCMP(
			ADR(usedStringToCheck[character]),
			usedSearchString, 
			lengthSearchString
		) = CNM_ReturnTypes.ComparationResult.EQUAL
	) THEN
		THIS^.freeMemory(usedStringToCheck, ignoreCases);
		THIS^.freeMemory(usedSearchString, ignoreCases);		
		RETURN; //assert is true
	END_IF; 
END_FOR

THIS^.assertionWasWrong(message, THIS^.getDebugInfo('contains'));
THIS^.freeMemory(usedStringToCheck, ignoreCases);
THIS^.freeMemory(usedSearchString, ignoreCases);
END_METHOD

(*

short summary
=================
This assertion method checks if the current string ``stringToCheck`` doesn't contain the search string ``searchString``.
Processed strings must be in Windows-1252 or Windows-1251 encoding

.. attention:: 
	All strings are handled as null-terminated byte streams

.. <legal notes>

legal notes
=================
| SPDX-FileCopyrightText: © 2024 ekvip automation GmbH <info@ekvip.de>
| SPDX-License-Identifier: Apache-2.0
| For details check: Apache-2.0_

.. _Apache-2.0: https://www.apache.org/licenses/LICENSE-2.0

.. </legal notes>

parameters
=================

*)

METHOD containsNo : IWindows125xStringPointerAssertions
VAR_INPUT
	(* current string to check *)
	stringToCheck	:POINTER TO BYTE;
	(* string must be found in ``stringToCheck`` *)
	searchString	:POINTER TO BYTE;
	(* ``TRUE`` means ignore cases; ``FALSE`` means that cases must be equal too *)
	ignoreCases		:BOOL;
	(* message if the assertion is false *)
	message			:AssertMessage;
END_VAR
VAR
	(* length of current string to check *)
	lenghtStringToCheck	:UDINT;
	(* length of ``searchString`` *)
	lengthSearchString	:UDINT;
	(* string address we use to compare, if it's case sensitive it's equal to ``stringToCheck`` *)
	usedStringToCheck	:POINTER TO BYTE;
	(* seacrch string address we use to compare, if it's case sensitive it's equal to ``searchString`` *)
	usedSearchString	:POINTER TO BYTE;
	(* character index for the comperation *)
	character			:UDINT;
END_VAR
containsNo := THIS^;

lenghtStringToCheck := THIS^.getStringLength(stringToCheck);
lengthSearchString := THIS^.getStringLength(searchString);

IF (
	NOT THIS^.isContainsNoCheckNecessary(
		stringToCheck		:= stringToCheck,
		searchString		:= searchString,
		lenghtStringToCheck	:= lenghtStringToCheck,
		lengthSearchString	:= lengthSearchString,
		additionalText		:= THIS^.getDebugInfo('containsNo'),
		message				:= message
	)
) THEN
	RETURN;
END_IF

usedStringToCheck := THIS^.getNewUpperCaseString(stringToCheck, lenghtStringToCheck, ignoreCases);
usedSearchString := THIS^.getNewUpperCaseString(searchString, lengthSearchString, ignoreCases);

FOR (character := 0) TO (lenghtStringToCheck - lengthSearchString) BY 1 DO
	IF (Tc2_System.MEMCMP(
			ADR(usedStringToCheck[character]),
			usedSearchString, 
			lengthSearchString
		) = CNM_ReturnTypes.ComparationResult.EQUAL
	) THEN
		THIS^.assertionWasWrong(message, THIS^.getDebugInfo('containsNo'));
		THIS^.freeMemory(usedStringToCheck, ignoreCases);
		THIS^.freeMemory(usedSearchString, ignoreCases);		
		RETURN;
	END_IF; 
END_FOR

THIS^.freeMemory(usedStringToCheck, ignoreCases);
THIS^.freeMemory(usedSearchString, ignoreCases);
END_METHOD

(*

short summary
=================
This assertion method checks if the current string ``stringToCheck`` ends with the string ``end``.
Processed strings must be in Windows-1252 or Windows-1251 encoding

.. attention:: 
	All strings are handled as null-terminated byte streams

.. <legal notes>

legal notes
=================
| SPDX-FileCopyrightText: © 2024 ekvip automation GmbH <info@ekvip.de>
| SPDX-License-Identifier: Apache-2.0
| For details check: Apache-2.0_

.. _Apache-2.0: https://www.apache.org/licenses/LICENSE-2.0

.. </legal notes>

parameters
=================

*)

METHOD endsWith : IWindows125xStringPointerAssertions
VAR_INPUT
	(* current string to check *)
	stringToCheck	:POINTER TO BYTE;
	(* string must be the end of ``stringToCheck`` *)
	end				:POINTER TO BYTE;
	(* ``TRUE`` means ignore cases; ``FALSE`` means that cases must be equal too *)
	ignoreCases		:BOOL;
	(* ``TRUE`` means truncation of spaces on the right side of ``stringToCheck``*)
	trimRight		:BOOL;
	(* message if the assertion is false *)
	message			:AssertMessage;
END_VAR
VAR
	(* length of current string to check *)
	lenghtStringToCheck	:UDINT;
	(* length of ``end`` *)
	lengthOfEnd			:UDINT;
	(* string address we use to compare, if it's case sensitive it's equal to ``stringToCheck`` *)
	usedStringToCheck	:POINTER TO BYTE;
	(* seacrch string address we use to compare, if it's case sensitive it's equal to ``end`` *)
	usedEndString		:POINTER TO BYTE;
END_VAR
endsWith := THIS^;

lenghtStringToCheck := THIS^.getStringLength(stringToCheck);
lengthOfEnd := THIS^.getStringLength(end);

THIS^.trimRight(stringToCheck, lenghtStringToCheck, trimRight);

IF (
	NOT THIS^.isContainsCheckNecessary(
		stringToCheck		:= stringToCheck,
		searchString		:= end,
		lenghtStringToCheck	:= lenghtStringToCheck,
		lengthSearchString	:= lengthOfEnd,
		additionalText		:= THIS^.getDebugInfo('endsWith'),
		message				:= message
	)
) THEN
	RETURN;
END_IF

usedStringToCheck := THIS^.getNewUpperCaseString(stringToCheck, lenghtStringToCheck, ignoreCases);
usedEndString := THIS^.getNewUpperCaseString(end, lengthOfEnd, ignoreCases);

IF (Tc2_System.MEMCMP(
		ADR(usedStringToCheck[lenghtStringToCheck - lengthOfEnd]),
		usedEndString, 
		lengthOfEnd
	) <> CNM_ReturnTypes.ComparationResult.EQUAL
) THEN
	THIS^.assertionWasWrong(message, THIS^.getDebugInfo('endsWith'));
END_IF;

THIS^.freeMemory(usedStringToCheck, ignoreCases);
THIS^.freeMemory(usedEndString, ignoreCases);
END_METHOD

(*

short summary
=================
This method is used to free allocated memory if needed

.. <legal notes>

legal notes
=================
| SPDX-FileCopyrightText: © 2024 ekvip automation GmbH <info@ekvip.de>
| SPDX-License-Identifier: Apache-2.0
| For details check: Apache-2.0_

.. _Apache-2.0: https://www.apache.org/licenses/LICENSE-2.0

.. </legal notes>

parameters
=================

*)

METHOD PROTECTED freeMemory
VAR_INPUT
	(* start address of the memory to free *)
	stringAddress	:POINTER TO BYTE;
	(* ``TRUE`` means free the memory, ``FALSE`` means do not free the memory *)
	freeMemory		:BOOL;
END_VAR
IF (freeMemory) THEN
	__DELETE(stringAddress);
END_IF
END_METHOD

(*

short summary
=================
this methods copy a string and returns the start address of new string,
all small letters are capitalized in the new string.

.. <legal notes>

legal notes
=================
| SPDX-FileCopyrightText: © 2024 ekvip automation GmbH <info@ekvip.de>
| SPDX-License-Identifier: Apache-2.0
| For details check: Apache-2.0_

.. _Apache-2.0: https://www.apache.org/licenses/LICENSE-2.0

.. </legal notes>

parameters
=================
:return: start address of a string. 
If ``createNewUpperCaseString`` is ``TRUE`` then it's a new string

*)

METHOD PROTECTED getNewUpperCaseString :POINTER TO BYTE; 
VAR_INPUT
	(* start address of the string to copy and capitalize *)
	stringAddress				:POINTER TO BYTE;
	(* length of the string ``stringAddress`` *)
	stringLength				:UDINT;
	(* 
	``TRUE means meake a copy and capitalize it, 
	``FALSE`` means return just ``stringAddress``
	and do nothing else
	*)
	createNewUpperCaseString	:BOOL;
END_VAR
IF (createNewUpperCaseString) THEN
	getNewUpperCaseString := THIS^.getStringCopy(stringAddress, stringLength);
	THIS^.upperCase(getNewUpperCaseString, stringLength);
ELSE
	getNewUpperCaseString := stringAddress;
END_IF
END_METHOD

(*

short summary
=================
this methods copy a string and returns the start address of new string

.. <legal notes>

legal notes
=================
| SPDX-FileCopyrightText: © 2024 ekvip automation GmbH <info@ekvip.de>
| SPDX-License-Identifier: Apache-2.0
| For details check: Apache-2.0_

.. _Apache-2.0: https://www.apache.org/licenses/LICENSE-2.0

.. </legal notes>

parameters
=================
:return: start address of the string copy

*)

METHOD PROTECTED getStringCopy :POINTER TO BYTE
VAR_INPUT
	(* string to copy *)
	stringAddress		:POINTER TO BYTE;
	(* length of the string *)
	stringLength		:UDINT;
END_VAR
getStringCopy := __NEW(BYTE, stringLength);
IF (getStringCopy <> 0) THEN
	Tc2_System.MEMCPY(
		destAddr := getStringCopy,
		srcAddr := stringAddress,
		n := stringLength
	);
END_IF
END_METHOD

(*

short summary
=================
this methods returns the length of a null-terminated string in bytes

.. attention:: 
	All strings are handled as null-terminated byte streams.

.. <legal notes>

legal notes
=================
| SPDX-FileCopyrightText: © 2024 ekvip automation GmbH <info@ekvip.de>
| SPDX-License-Identifier: Apache-2.0
| For details check: Apache-2.0_

.. _Apache-2.0: https://www.apache.org/licenses/LICENSE-2.0

.. </legal notes>

parameters
=================
:return: length of the string

*)

METHOD PROTECTED getStringLength :UDINT
VAR_INPUT
	(* Start address of the string for which the length is to be determined *)
	stringAddress	:POINTER TO BYTE;
END_VAR
VAR CONSTANT
	(* the end of string marker *)
	END_OF_STRING	:BYTE := 16#00;
END_VAR
IF (stringAddress = 0) THEN
	RETURN;
END_IF

WHILE (stringAddress[getStringLength] <> END_OF_STRING) DO
	getStringLength := getStringLength + 1;
END_WHILE
END_METHOD

(*

short summary
=================
this methods checks if a windows-1252 or a windows-1251 character is a whitespace character

.. <legal notes>

legal notes
=================
| SPDX-FileCopyrightText: © 2024 ekvip automation GmbH <info@ekvip.de>
| SPDX-License-Identifier: Apache-2.0
| For details check: Apache-2.0_

.. _Apache-2.0: https://www.apache.org/licenses/LICENSE-2.0

.. </legal notes>

parameters
=================
:return: ``TRUE`` means ``character`` is whitespace,
``FALSE`` means ``character`` is no whitespace 

*)

METHOD PROTECTED isCharWhiteSpace :BOOL
VAR_INPUT
	(* character to check if it's whitespace *)
	character	:BYTE;
END_VAR
VAR CONSTANT
	SPACE			:BYTE := 16#20;
	HORIZONTAL_TAB	:BYTE := 16#09;
	LINE_FEED		:BYTE := 16#0A;
	VERTICAL_TAB	:BYTE := 16#0B;
	FROM_FEED		:BYTE := 16#0C;
	CARRIAGE_RETURN	:BYTE := 16#0D;
END_VAR
CASE character OF
	HORIZONTAL_TAB .. CARRIAGE_RETURN,
	SPACE:
		isCharWhiteSpace := TRUE;
	ELSE
		isCharWhiteSpace := FALSE;	
END_CASE
END_METHOD

(*

short summary
=================
This assertion method checks if the current string ``stringToCheck`` is equal to ``expected``.
Processed strings must be in Windows-1252 or Windows-1251 encoding

.. attention:: 
	All strings are handled as null-terminated byte streams

.. <legal notes>

legal notes
=================
| SPDX-FileCopyrightText: © 2024 ekvip automation GmbH <info@ekvip.de>
| SPDX-License-Identifier: Apache-2.0
| For details check: Apache-2.0_

.. _Apache-2.0: https://www.apache.org/licenses/LICENSE-2.0

.. </legal notes>

parameters
=================

*)

METHOD isEqualTo : IWindows125xStringPointerAssertions
VAR_INPUT
	(* current string to check *)
	stringToCheck	:POINTER TO BYTE;
	(* ``stringToCheck`` must be equal to expected *)
	expected		:POINTER TO BYTE;
	(* ``TRUE`` means ignore cases; ``FALSE`` means that cases must be equal too *)
	ignoreCases		:BOOL;
	(* message if the assertion is false *)
	message			:AssertMessage;
END_VAR
VAR
	(* length of current string to check *)
	lenghtStringToCheck		:UDINT;
	(* length of ``expected`` *)
	lengthExpectedString	:UDINT;
	(* string address we use to compare, if it's case sensitive it's equal to ``stringToCheck`` *)
	usedStringToCheck		:POINTER TO BYTE;
	(* seacrch string address we use to compare, if it's case sensitive it's equal to ``expected`` *)
	usedExpectedString		:POINTER TO BYTE;
END_VAR
VAR CONSTANT
	(* length of an empty string to avoid Tc2_System.MEMCMP with length 0 *)
	EMPTY_STRING_LENGTH		:UDINT := 0;
END_VAR
isEqualTo := THIS^;

lenghtStringToCheck := THIS^.getStringLength(stringToCheck);
lengthExpectedString := THIS^.getStringLength(expected);

IF lenghtStringToCheck <> lengthExpectedString THEN
	THIS^.assertionWasWrong(message, THIS^.getDebugInfo('isEqualTo'));
	RETURN;
ELSIF (lengthExpectedString = EMPTY_STRING_LENGTH) THEN
	RETURN;
END_IF

usedStringToCheck := THIS^.getNewUpperCaseString(stringToCheck, lenghtStringToCheck, ignoreCases);
usedExpectedString := THIS^.getNewUpperCaseString(expected, lengthExpectedString, ignoreCases);

IF (Tc2_System.MEMCMP(
		usedStringToCheck,
		usedExpectedString, 
		lengthExpectedString
	) <> CNM_ReturnTypes.ComparationResult.EQUAL
) THEN
	THIS^.assertionWasWrong(message, THIS^.getDebugInfo('isEqualTo'));
END_IF;

THIS^.freeMemory(usedStringToCheck, ignoreCases);
THIS^.freeMemory(usedExpectedString, ignoreCases);
END_METHOD

(*

short summary
=================
This assertion method checks if the current string ``stringToCheck`` is not equal to ``unexpected``.
Processed strings must be in Windows-1252 or Windows-1251 encoding

.. attention:: 
	All strings are handled as null-terminated byte streams

.. <legal notes>

legal notes
=================
| SPDX-FileCopyrightText: © 2024 ekvip automation GmbH <info@ekvip.de>
| SPDX-License-Identifier: Apache-2.0
| For details check: Apache-2.0_

.. _Apache-2.0: https://www.apache.org/licenses/LICENSE-2.0

.. </legal notes>

parameters
=================

*)

METHOD isNotEqualTo : IWindows125xStringPointerAssertions
VAR_INPUT
	(* current string to check *)
	stringToCheck	:POINTER TO BYTE;
	(* ``stringToCheck`` must be not equal to expected *)
	unexpected		:POINTER TO BYTE;
	(* ``TRUE`` means ignore cases; ``FALSE`` means that cases must be equal too *)
	ignoreCases		:BOOL;
	(* message if the assertion is false *)
	message			:AssertMessage;
END_VAR
VAR
	(* length of current string to check *)
	lenghtStringToCheck		:UDINT;
	(* length of ``unexpected`` *)
	lengthUnexpectedString	:UDINT;
	(* string address we use to compare, if it's case sensitive it's equal to ``stringToCheck`` *)
	usedStringToCheck		:POINTER TO BYTE;
	(* seacrch string address we use to compare, if it's case sensitive it's equal to ``expected`` *)
	usedUnexpectedString	:POINTER TO BYTE;
END_VAR
VAR CONSTANT
	(* length of an empty string to avoid Tc2_System.MEMCMP with length 0 *)
	EMPTY_STRING_LENGTH		:UDINT := 0;
END_VAR
isNotEqualTo := THIS^;

lenghtStringToCheck := THIS^.getStringLength(stringToCheck);
lengthUnexpectedString := THIS^.getStringLength(unexpected);

IF lenghtStringToCheck = EMPTY_STRING_LENGTH AND_THEN lengthUnexpectedString = EMPTY_STRING_LENGTH THEN
	THIS^.assertionWasWrong(message, THIS^.getDebugInfo('isNotEqualTo'));
	RETURN;
END_IF

usedStringToCheck := THIS^.getNewUpperCaseString(stringToCheck, lenghtStringToCheck, ignoreCases);
usedUnexpectedString := THIS^.getNewUpperCaseString(unexpected, lengthUnexpectedString, ignoreCases);

IF (Tc2_System.MEMCMP(
		usedStringToCheck,
		usedUnexpectedString, 
		lengthUnexpectedString
	) = CNM_ReturnTypes.ComparationResult.EQUAL
) THEN
	THIS^.assertionWasWrong(message, THIS^.getDebugInfo('isNotEqualTo'));
END_IF;

THIS^.freeMemory(usedStringToCheck, ignoreCases);
THIS^.freeMemory(usedUnexpectedString, ignoreCases);
END_METHOD

(*

short summary
=================
This assertion method checks if the current string ``stringToCheck`` length is equal to ``expectedLength``.
Processed strings must be in Windows-1252 or Windows-1251 encoding

.. attention:: 
	All strings are handled as null-terminated byte streams

.. <legal notes>

legal notes
=================
| SPDX-FileCopyrightText: © 2024 ekvip automation GmbH <info@ekvip.de>
| SPDX-License-Identifier: Apache-2.0
| For details check: Apache-2.0_

.. _Apache-2.0: https://www.apache.org/licenses/LICENSE-2.0

.. </legal notes>

parameters
=================

*)

METHOD lenghtIsExact : IWindows125xStringPointerAssertions
VAR_INPUT
	(* current string to check *)
	stringToCheck	:POINTER TO BYTE;
	(* expected length of ``stringToCheck`` *)
	expectedLength	:UDINT;
	(* message if the assertion is false *)
	message			:AssertMessage;
END_VAR
lenghtIsExact := THIS^;

IF (THIS^.getStringLength(stringToCheck) <> expectedLength) THEN
	THIS^.assertionWasWrong(message, THIS^.getDebugInfo('lenghtIsExact'));
END_IF
END_METHOD

(*

short summary
=================
This assertion method checks if the current string ``stringToCheck`` length is equal or less than to ``maxLength``.
Processed strings must be in Windows-1252 or Windows-1251 encoding

.. attention:: 
	All strings are handled as null-terminated byte streams

.. <legal notes>

legal notes
=================
| SPDX-FileCopyrightText: © 2024 ekvip automation GmbH <info@ekvip.de>
| SPDX-License-Identifier: Apache-2.0
| For details check: Apache-2.0_

.. _Apache-2.0: https://www.apache.org/licenses/LICENSE-2.0

.. </legal notes>

parameters
=================

*)

METHOD lenghtIsMax : IWindows125xStringPointerAssertions
VAR_INPUT
	(* current string to check *)
	stringToCheck	:POINTER TO BYTE;
	(* upper limit of the length of ``stringToCheck`` *)
	maxLength		:UDINT;
	(* message if the assertion is false *)
	message			:AssertMessage;
END_VAR
lenghtIsMax := THIS^;

IF (THIS^.getStringLength(stringToCheck) > maxLength) THEN
	THIS^.assertionWasWrong(message, THIS^.getDebugInfo('lenghtIsMax'));
END_IF
END_METHOD

(*

short summary
=================
This assertion method checks if the current string ``stringToCheck`` length is equal or grater than to ``minLength``.
Processed strings must be in Windows-1252 or Windows-1251 encoding

.. attention:: 
	All strings are handled as null-terminated byte streams

.. <legal notes>

legal notes
=================
| SPDX-FileCopyrightText: © 2024 ekvip automation GmbH <info@ekvip.de>
| SPDX-License-Identifier: Apache-2.0
| For details check: Apache-2.0_

.. _Apache-2.0: https://www.apache.org/licenses/LICENSE-2.0

.. </legal notes>

parameters
=================

*)

METHOD lenghtIsMin : IWindows125xStringPointerAssertions
VAR_INPUT
	(* current string to check *)
	stringToCheck	:POINTER TO BYTE;
	(* lower limit of the length of ``stringToCheck`` *)
	minLength		:UDINT;
	(* message if the assertion is false *)
	message			:AssertMessage;
END_VAR
lenghtIsMin := THIS^;

IF (THIS^.getStringLength(stringToCheck) < minLength) THEN
	THIS^.assertionWasWrong(message, THIS^.getDebugInfo('lenghtIsMin'));
END_IF
END_METHOD

(*

short summary
=================
This assertion method checks if the current string ``stringToCheck`` length is between ``minLenght`` and ``maxLenght``.
Processed strings must be in Windows-1252 or Windows-1251 encoding

.. attention:: 
	All strings are handled as null-terminated byte streams

.. <legal notes>

legal notes
=================
| SPDX-FileCopyrightText: © 2024 ekvip automation GmbH <info@ekvip.de>
| SPDX-License-Identifier: Apache-2.0
| For details check: Apache-2.0_

.. _Apache-2.0: https://www.apache.org/licenses/LICENSE-2.0

.. </legal notes>

parameters
=================

*)

METHOD lengthIsBetween : IWindows125xStringPointerAssertions
VAR_INPUT
	(* current string to check *)
	stringToCheck	:POINTER TO BYTE;
	(* lower limit of the string length *)
	minLenght		:UDINT;
	(* upper limit of the string length *)
	maxLenght		:UDINT;
	(* message if the assertion is false *)
	message			:AssertMessage;
END_VAR
VAR
	(* length of ``stringToCheck`` *)
	lenghtStringToCheck	:UDINT;
END_VAR
lengthIsBetween := THIS^;

IF minLenght > maxLenght THEN
	THIS^.assertionWasWrong(message, THIS^.getDebugInfo('lengthIsBetween'));
	RETURN;
END_IF

lenghtStringToCheck := THIS^.getStringLength(stringToCheck);

IF lenghtStringToCheck < minLenght OR_ELSE lenghtStringToCheck > maxLenght THEN
	THIS^.assertionWasWrong(message, THIS^.getDebugInfo('lengthIsBetween'));
END_IF;
END_METHOD

(*

short summary
=================
This assertion method checks if the current string ``stringToCheck`` starts with string ``start``.
Processed strings must be in Windows-1252 or Windows-1251 encoding

.. attention:: 
	All strings are handled as null-terminated byte streams

.. <legal notes>

legal notes
=================
| SPDX-FileCopyrightText: © 2024 ekvip automation GmbH <info@ekvip.de>
| SPDX-License-Identifier: Apache-2.0
| For details check: Apache-2.0_

.. _Apache-2.0: https://www.apache.org/licenses/LICENSE-2.0

.. </legal notes>

parameters
=================

*)

METHOD startsWith : IWindows125xStringPointerAssertions
VAR_INPUT
	(* current string to check *)
	stringToCheck	:POINTER TO BYTE;
	(* expected start of ``stringToCheck`` *)
	start			:POINTER TO BYTE;
	(* ``TRUE`` means ignore cases; ``FALSE`` means that cases must be equal too *)
	ignoreCases		:BOOL;
	(* ``TRUE`` means truncation of spaces on the left side of ``stringToCheck``*)
	trimLeft		:BOOL;
	(* message if the assertion is false *)
	message			:AssertMessage;
END_VAR
VAR
	(* length of current string to check *)
	lenghtStringToCheck	:UDINT;
	(* length of ``start`` *)
	lengthOfStart		:UDINT;
	(* string address we use to compare, if it's case sensitive it's equal to ``stringToCheck`` *)
	usedStringToCheck	:POINTER TO BYTE;
	(* seacrch string address we use to compare, if it's case sensitive it's equal to ``start`` *)
	usedStartString		:POINTER TO BYTE;
END_VAR
startsWith := THIS^;

lenghtStringToCheck := THIS^.getStringLength(stringToCheck);
lengthOfStart := THIS^.getStringLength(start);

THIS^.trimLeft(stringToCheck, lenghtStringToCheck, trimLeft);

IF (
	NOT THIS^.isContainsCheckNecessary(
		stringToCheck		:= stringToCheck,
		searchString		:= start,
		lenghtStringToCheck	:= lenghtStringToCheck,
		lengthSearchString	:= lengthOfStart,
		additionalText		:= THIS^.getDebugInfo('startsWith'),
		message				:= message
	)
) THEN
	RETURN;
END_IF

usedStringToCheck := THIS^.getNewUpperCaseString(stringToCheck, lenghtStringToCheck, ignoreCases);
usedStartString := THIS^.getNewUpperCaseString(start, lengthOfStart, ignoreCases);

IF (Tc2_System.MEMCMP(
		usedStringToCheck,
		usedStartString, 
		lengthOfStart
	) <> CNM_ReturnTypes.ComparationResult.EQUAL
) THEN
	THIS^.assertionWasWrong(message, THIS^.getDebugInfo('startsWith'));
END_IF;

THIS^.freeMemory(usedStringToCheck, ignoreCases);
THIS^.freeMemory(usedStartString, ignoreCases);
END_METHOD

(*

short summary
=================
This method is used to remove the whitespace from the start of the string.
It does not really remove it, it just moves the start address and decreases
the string length

.. <legal notes>

legal notes
=================
| SPDX-FileCopyrightText: © 2024 ekvip automation GmbH <info@ekvip.de>
| SPDX-License-Identifier: Apache-2.0
| For details check: Apache-2.0_

.. _Apache-2.0: https://www.apache.org/licenses/LICENSE-2.0

.. </legal notes>

parameters
=================

*)

METHOD PROTECTED trimLeft
VAR_IN_OUT
	(* start address of the string *)
	stringAddress	:POINTER TO BYTE;
	(* length of the string ``stringAddress`` *)
	stringLength	:UDINT;
END_VAR
VAR_INPUT
	(* ``TRUE`` means remove the whitespace, ``FALSE`` means do not remove the whitespace *)
	trimString		:BOOL;
END_VAR
VAR
	(* index of the current character *)
	character		:UDINT;
	(* counter of the whitspace characters *)
	whitespaceCount	:UDINT;
END_VAR
IF (stringAddress = 0 OR_ELSE stringLength <= 0 OR_ELSE NOT trimString) THEN
	RETURN;
END_IF

FOR character := 0 TO stringLength - 1 DO
	IF (THIS^.isCharWhiteSpace(stringAddress[character])) THEN
		whitespaceCount := whitespaceCount + 1;
	ELSE
		EXIT;
	END_IF
END_FOR

stringAddress := ADR(stringAddress[whitespaceCount]);
stringLength := stringLength - whitespaceCount;
END_METHOD

(*

short summary
=================
This method is used to remove the whitespace from the end of the string.
It does not really remove it, it just decreases the string length.

.. <legal notes>

legal notes
=================
| SPDX-FileCopyrightText: © 2024 ekvip automation GmbH <info@ekvip.de>
| SPDX-License-Identifier: Apache-2.0
| For details check: Apache-2.0_

.. _Apache-2.0: https://www.apache.org/licenses/LICENSE-2.0

.. </legal notes>

parameters
=================

*)

METHOD PROTECTED trimRight
VAR_INPUT
	(* start address of the string *)
	stringAddress	:POINTER TO BYTE;
END_VAR
VAR_IN_OUT
	(* length of the string ``stringAddress`` *)
	stringLength	:UDINT;
END_VAR
VAR_INPUT
	(* ``TRUE`` means remove the whitespace, ``FALSE`` means do not remove the whitespace *)
	trimString		:BOOL;
END_VAR
VAR
	(* index of the current character *)
	character	:LINT;
END_VAR
IF stringAddress = 0 OR_ELSE stringLength <= 0 OR_ELSE NOT trimString THEN
	RETURN;
END_IF

FOR character := (stringLength-1) TO 0 BY -1 DO
	IF (THIS^.isCharWhiteSpace(stringAddress[character])) THEN
		stringLength := stringLength-1;
	ELSE
		RETURN;
	END_IF
END_FOR
END_METHOD

(*

short summary
=================
This method converts the lowercase letters in an 8 bit windows-1252 or windows-1251
string to uppercase letters.

.. attention:: 
	All strings are handled as null-terminated byte streams.

.. <legal notes>

legal notes
=================
| SPDX-FileCopyrightText: © 2024 ekvip automation GmbH <info@ekvip.de>
| SPDX-License-Identifier: Apache-2.0
| For details check: Apache-2.0_

.. _Apache-2.0: https://www.apache.org/licenses/LICENSE-2.0

.. </legal notes>

parameters
=================

*)

METHOD PROTECTED upperCase
VAR_INPUT
	(* string to ucase *)
	stringAddress	:POINTER TO BYTE;
	(* length of the string *)
	stringLength	:UDINT;
END_VAR
IF (stringAddress = 0) THEN
	RETURN;
END_IF

CASE Tc2_Utilities.GLOBAL_SBCS_TABLE OF
	Tc2_Utilities.E_SBCSType.eSBCS_WesternEuropean:
		upperCase1252(stringAddress, stringLength);
		
	Tc2_Utilities.E_SBCSType.eSBCS_CentralEuropean:
		upperCase1251(stringAddress, stringLength);
END_CASE
END_METHOD

(*

short summary
=================
This method converts the lowercase letters in an 8 bit windows-1251
string to uppercase letters.

.. attention:: 
	All strings are handled as null-terminated byte streams.

.. <legal notes>

legal notes
=================
| SPDX-FileCopyrightText: © 2024 ekvip automation GmbH <info@ekvip.de>
| SPDX-License-Identifier: Apache-2.0
| For details check: Apache-2.0_

.. _Apache-2.0: https://www.apache.org/licenses/LICENSE-2.0

.. </legal notes>

parameters
=================

*)

METHOD PROTECTED upperCase1251
VAR_INPUT
	(* string to ucase *)
	stringAddress		:POINTER TO BYTE;
	(* length of the string *)
	stringLength		:UDINT;
END_VAR
VAR
	(* index of the current character *)
	character			:UDINT := 0;
END_VAR
VAR CONSTANT
	(* NUL: $00 *)
	END_OF_STRING							:BYTE := 16#00;
	(* a *)                             	
	LOWERCASE_A								:BYTE := 16#61;
	(* z *)                             	
	LOWERCASE_Z								:BYTE := 16#7A;	
	(* а *)
	LOWERCASE_CYRILLIC_A					:BYTE := 16#E0;
	(* я *)
	LOWERCASE_CYRILLIC_YA					:BYTE := 16#FF;
	
	(* ђ *)
	LOWERCASE_CYRILLIC_DJE					:BYTE := 16#90;
	(* љ *)
	LOWERCASE_CYRILLIC_LJE					:BYTE := 16#9A;
	(* њ *)
	LOWERCASE_CYRILLIC_NJE					:BYTE := 16#9C;	
	(* џ *)
	LOWERCASE_CYRILLIC_DZHE					:BYTE := 16#9F;
	(* ё *)
	LOWERCASE_CYRILLIC_IO					:BYTE := 16#B8;
	(* є *)
	LOWERCASE_CYRILLIC_UKRAINIAN_IE			:BYTE := 16#BA;
	(* ї *)
	LOWERCASE_CYRILLIC_YI					:BYTE := 16#BF;

	(* ў *)
	LOWERCASE_CYRILLIC_SHORT_U				:BYTE := 16#A2;
	(* i *)
	LOWERCASE_CYRILLIC_UKRAINIAN_I			:BYTE := 16#B3;
	(* ѕ *)
	LOWERCASE_CYRILLIC_DZE					:BYTE := 16#BE;
	
	(* ѓ *)
	LOWERCASE_CYRILLIC_GJE					:BYTE := 16#83;
	
	(* ґ *)
	LOWERCASE_CYRILLIC_GHE_WITH_UPTURN		:BYTE := 16#B4;
	
	(* ј *)
	LOWERCASE_CYRILLIC_JE					:BYTE := 16#19;
END_VAR
WHILE stringAddress[character] <> END_OF_STRING AND_THEN character <= stringLength DO
	CASE stringAddress[character] OF
		LOWERCASE_A..LOWERCASE_Z,
		LOWERCASE_CYRILLIC_A..LOWERCASE_CYRILLIC_YA:
			stringAddress[character] := stringAddress[character] - 16#20;
		LOWERCASE_CYRILLIC_DJE,
		LOWERCASE_CYRILLIC_LJE,
		LOWERCASE_CYRILLIC_NJE..LOWERCASE_CYRILLIC_DZHE,
		LOWERCASE_CYRILLIC_IO,
		LOWERCASE_CYRILLIC_UKRAINIAN_IE,
		LOWERCASE_CYRILLIC_YI:
			stringAddress[character] := stringAddress[character] - 16#10;
		LOWERCASE_CYRILLIC_SHORT_U,
		LOWERCASE_CYRILLIC_UKRAINIAN_I,
		LOWERCASE_CYRILLIC_DZE:
			stringAddress[character] := 16#01;
		LOWERCASE_CYRILLIC_GJE:
			stringAddress[character] := 16#02;
		LOWERCASE_CYRILLIC_GHE_WITH_UPTURN:
			stringAddress[character] := 16#0F;
		LOWERCASE_CYRILLIC_JE:
			stringAddress[character] := 16#0F;
	END_CASE
	
	character := character + 1;
END_WHILE
END_METHOD

(*

short summary
=================
This method converts the lowercase letters in an 8 bit windows-1252 
string to uppercase letters.

.. attention:: 
	All strings are handled as null terminated byte streams.

.. <legal notes>

legal notes
=================
| SPDX-FileCopyrightText: © 2024 ekvip automation GmbH <info@ekvip.de>
| SPDX-License-Identifier: Apache-2.0
| For details check: Apache-2.0_

.. _Apache-2.0: https://www.apache.org/licenses/LICENSE-2.0

.. </legal notes>

parameters
=================

*)

METHOD PROTECTED upperCase1252
VAR_INPUT
	(* string to ucase *)
	stringAddress		:POINTER TO BYTE;
	(* length of the string *)
	stringLength		:UDINT;
END_VAR
VAR
	(* index of the current character *)
	character			:UDINT := 0;
END_VAR
VAR CONSTANT
	(* NUL: $00 *)
	END_OF_STRING							:BYTE := 16#00;
	(* a *)                             	
	LOWERCASE_A								:BYTE := 16#61;
	(* z *)                             	
	LOWERCASE_Z								:BYTE := 16#7A;
	(* ß *)                             	
	LOWERCASE_SHARP_S						:BYTE := 16#DF;
	(* ÿ *)                             	
	LOWERCASE_Y_WITH_DIAERESIS				:BYTE := 16#FF;
	(* Ÿ *)                             	
	UPPERCASE_Y_WITH_DIAERESIS				:BYTE := 16#9F;
	(* à *)                             	
	LOWERCASE_A_WITH_GRAVE					:BYTE := 16#E0;
	(* ö *)                             	
	LOWERCASE_O_WITH_DIAERESIS				:BYTE := 16#F6;
	(* ø *)                             	
	LOWERCASE_O_WITH_SLASH					:BYTE := 16#F8;
	(* þ *)                             	
	LOWERCASE_THORN							:BYTE := 16#FE;
	(* š *)                             	
	LOWERCASE_S_WITH_CARON					:BYTE := 16#9A;
	(* œ *)                             	
	LOWERCASE_OE							:BYTE := 16#9C;
	(* ž *)                             	
	LOWERCASE_Z_WITH_CARON					:BYTE := 16#9E;
	(* difference between lowercase and uppercase except for š,œ and ž *)
	DIFFERENCE_LOWERCASE_UPPERCASE			:BYTE := 16#20;
	(* for š,œ and ž the difference between lowercase and uppercase *)
	DIFFERENCE_LOWERCASE_UPPERCASE_SPECIAL	:BYTE := 16#10;
END_VAR
WHILE stringAddress[character] <> END_OF_STRING AND_THEN character <= stringLength DO
	CASE stringAddress[character] OF
		LOWERCASE_A..LOWERCASE_Z,
		LOWERCASE_A_WITH_GRAVE..LOWERCASE_O_WITH_DIAERESIS,
		LOWERCASE_O_WITH_SLASH..LOWERCASE_THORN:
			stringAddress[character] := stringAddress[character] - DIFFERENCE_LOWERCASE_UPPERCASE;
		LOWERCASE_S_WITH_CARON,
		LOWERCASE_OE,
		LOWERCASE_Z_WITH_CARON:
			stringAddress[character] := stringAddress[character] - DIFFERENCE_LOWERCASE_UPPERCASE_SPECIAL;
		LOWERCASE_Y_WITH_DIAERESIS:
			stringAddress[character] := UPPERCASE_Y_WITH_DIAERESIS;
		LOWERCASE_SHARP_S:;//for ß do nothing, because there is no capital letter for it
	END_CASE
	
	character := character + 1;
END_WHILE
END_METHOD

END_FUNCTION_BLOCK

// ---- Assertor/Assertions/StringAssertion/WString/classes/utf16StringAssertions.TcPOU
(*

short summary
=================
This class provides assert statements for UTF-16 strings until 255 ``WORD`` length

.. <legal notes>

legal notes
=================
| SPDX-FileCopyrightText: © 2022 ekvip automation GmbH <info@ekvip.de>
| SPDX-License-Identifier: Apache-2.0
| For details check: Apache-2.0_

.. _Apache-2.0: https://www.apache.org/licenses/LICENSE-2.0

.. </legal notes>

methods and properties
=======================

*)

{attribute 'reflection'}
FUNCTION_BLOCK INTERNAL utf16StringAssertions EXTENDS AbstactAssertion IMPLEMENTS IUtf16StringAssertions
VAR
	(* class to handle the UTF-16 string assertions *)  
	assertion	:Utf16StringPointerAssertions();
END_VAR

(*

short summary
=================
This abstract property returns the class name of the concrete object, 
It's for debugging purpose

.. <legal notes>

legal notes
=================
| SPDX-FileCopyrightText: © 2022 ekvip automation GmbH <info@ekvip.de>
| SPDX-License-Identifier: Apache-2.0
| For details check: Apache-2.0_

.. _Apache-2.0: https://www.apache.org/licenses/LICENSE-2.0

.. </legal notes>

*)

PROPERTY className :CNM_AbstractObject.ClassName
GET
className := 'CNM_AssertionInterfaceLib.utf16StringAssertions';
END_GET
END_PROPERTY

(*

short summary
=================
This assertion method for UTF-16 strings checks if the current string ``stringToCheck`` contains the search string ``searchString``

.. <legal notes>

legal notes
=================
| SPDX-FileCopyrightText: © 2022 ekvip automation GmbH <info@ekvip.de>
| SPDX-License-Identifier: Apache-2.0
| For details check: Apache-2.0_

.. _Apache-2.0: https://www.apache.org/licenses/LICENSE-2.0

.. </legal notes>

parameters
=================

*)

METHOD contains
VAR_INPUT
	(* current string to check *)
	stringToCheck	:WSTRING(Tc2_System.MAX_STRING_LENGTH);
	(* string must be found in ``stringToCheck`` *)
	searchString	:WSTRING(Tc2_System.MAX_STRING_LENGTH);
	(* ``TRUE`` means ignore cases; ``FALSE`` means cases must be equal too *)
	ignoreCases		:BOOL;
	(* message if the assertion is false *)
	message			:AssertMessage;
END_VAR
THIS^.assertion.utf16Contains(
	stringToCheck 	:= ADR(stringToCheck),
	searchSTring 	:= ADR(searchString),
	ignoreCases 	:= ignoreCases,
	message 		:= message
);
END_METHOD

(*

short summary
=================
This assertion method for UTF-16 strings checks if the current string ``stringToCheck`` contains not the search string ``searchString``

.. <legal notes>

legal notes
=================
| SPDX-FileCopyrightText: © 2022 ekvip automation GmbH <info@ekvip.de>
| SPDX-License-Identifier: Apache-2.0
| For details check: Apache-2.0_

.. _Apache-2.0: https://www.apache.org/licenses/LICENSE-2.0

.. </legal notes>

parameters
=================

*)

METHOD containsNo
VAR_INPUT
	(* current string to check *)
	stringToCheck	:WSTRING(Tc2_System.MAX_STRING_LENGTH);
	(* string that must not be found in ``stringToCheck`` *)
	searchString	:WSTRING(Tc2_System.MAX_STRING_LENGTH);
	(* ``TRUE`` means ignore cases; ``FALSE`` means cases must be equal too *)
	ignoreCases		:BOOL;
	(* message if the assertion is false *)
	message			:AssertMessage;
END_VAR
THIS^.assertion.utf16ContainsNo(
	stringToCheck 	:= ADR(stringToCheck),
	searchSTring 	:= ADR(searchString),
	ignoreCases 	:= ignoreCases,
	message 		:= message
);
END_METHOD

(*

short summary
=================
This assertion method for UTF-16 strings checks if the current string ``stringToCheck`` ends with the string ``end``

.. attention:: 
	end of the string is **ALWAYS** the right side of the string 
	even for writings which written from right to left like Hebrew or Arabic

.. <legal notes>

legal notes
=================
| SPDX-FileCopyrightText: © 2022 ekvip automation GmbH <info@ekvip.de>
| SPDX-License-Identifier: Apache-2.0
| For details check: Apache-2.0_

.. _Apache-2.0: https://www.apache.org/licenses/LICENSE-2.0

.. </legal notes>

parameters
=================

*)

METHOD endsWith
VAR_INPUT
	(* current string to check *)
	stringToCheck	:WSTRING(Tc2_System.MAX_STRING_LENGTH);
	(* expected end of ``stringToCheck`` *)
	end				:WSTRING(Tc2_System.MAX_STRING_LENGTH);
	(* ``TRUE`` means ignore cases; ``FALSE`` means cases must be equal too *)
	ignoreCases		:BOOL;
	(* ``TRUE`` means truncation of spaces on the right side of ``stringToCheck``*)
	trim			:BOOL;
	(* message if the assertion is false *)
	message			:AssertMessage;
END_VAR
THIS^.assertion.utf16EndsWith(
	stringToCheck	:= ADR(stringToCheck),
	end				:= ADR(end),
	ignoreCases		:= ignoreCases,
	trim			:= trim,
	message			:= message
);
END_METHOD

(*

short summary
=================
This assertion method checks if the current string ``stringToCheck`` is empty

.. <legal notes>

legal notes
=================
| SPDX-FileCopyrightText: © 2022 ekvip automation GmbH <info@ekvip.de>
| SPDX-License-Identifier: Apache-2.0
| For details check: Apache-2.0_

.. _Apache-2.0: https://www.apache.org/licenses/LICENSE-2.0

.. </legal notes>

parameters
=================

*)

METHOD isEmpty
VAR_INPUT
	(* current string to check *)
	stringToCheck	:WSTRING(Tc2_System.MAX_STRING_LENGTH);
	(* message if the assertion is false *)
	message			:AssertMessage;
END_VAR
IF (stringToCheck <> "") THEN
	THIS^.assertionWasWrong(message, THIS^.getDebugInfo('isEmpty'));
END_IF
END_METHOD

(*

short summary
=================
This assertion method checks if the current string ``stringToCheck`` is equal to ``expected``

.. <legal notes>

legal notes
=================
| SPDX-FileCopyrightText: © 2022 ekvip automation GmbH <info@ekvip.de>
| SPDX-License-Identifier: Apache-2.0
| For details check: Apache-2.0_

.. _Apache-2.0: https://www.apache.org/licenses/LICENSE-2.0

.. </legal notes>

parameters
=================

*)

METHOD isEqualTo
VAR_INPUT
	(* current string to check *)
	stringToCheck	:WSTRING(Tc2_System.MAX_STRING_LENGTH);
	(* ``stringToCheck`` must be equal to expected *)
	expected		:WSTRING(Tc2_System.MAX_STRING_LENGTH);
	(* ``TRUE`` means ignore cases; ``FALSE`` means cases must be equal too *)
	ignoreCases		:BOOL;
	(* message if the assertion is false *)
	message			:AssertMessage;
END_VAR
THIS^.assertion.utf16IsEqualTo(
	stringToCheck	:= ADR(stringToCheck),
	expected		:= ADR(expected),
	ignoreCases		:= ignoreCases,
	message			:= message
);
END_METHOD

(*

short summary
=================
This assertion method checks if the current string ``stringToCheck`` is not empty

.. <legal notes>

legal notes
=================
| SPDX-FileCopyrightText: © 2022 ekvip automation GmbH <info@ekvip.de>
| SPDX-License-Identifier: Apache-2.0
| For details check: Apache-2.0_

.. _Apache-2.0: https://www.apache.org/licenses/LICENSE-2.0

.. </legal notes>

parameters
=================

*)

METHOD isNotEmpty
VAR_INPUT
	(* current string to check *)
	stringToCheck	:WSTRING(Tc2_System.MAX_STRING_LENGTH);
	(* message if the assertion is false *)
	message			:AssertMessage;
END_VAR
IF (stringToCheck = "") THEN
	THIS^.assertionWasWrong(message, THIS^.getDebugInfo('isNotEmpty'));
END_IF
END_METHOD

(*

short summary
=================
This assertion method checks if the current string ``stringToCheck`` is not equal to ``unexpected``

.. <legal notes>

legal notes
=================
| SPDX-FileCopyrightText: © 2022 ekvip automation GmbH <info@ekvip.de>
| SPDX-License-Identifier: Apache-2.0
| For details check: Apache-2.0_

.. _Apache-2.0: https://www.apache.org/licenses/LICENSE-2.0

.. </legal notes>

parameters
=================

*)

METHOD isNotEqualTo
VAR_INPUT
	(* current string to check *)
	stringToCheck	:WSTRING(Tc2_System.MAX_STRING_LENGTH);
	(* ``stringToCheck`` must be not equal to expected *)
	unexpected		:WSTRING(Tc2_System.MAX_STRING_LENGTH);
	(* ``TRUE`` means ignore cases; ``FALSE`` means cases must be equal too *)
	ignoreCases		:BOOL;
	(* message if the assertion is false *)
	message			:AssertMessage;
END_VAR
THIS^.assertion.utf16IsNotEqualTo(
	stringToCheck	:= ADR(stringToCheck),
	unexpected		:= ADR(unexpected),
	ignoreCases		:= ignoreCases,
	message			:= message
);
END_METHOD

(*

short summary
=================
This assertion method checks if the current string ``stringToCheck`` length
is between ``minLenght`` and ``maxLenght``

.. <legal notes>

legal notes
=================
| SPDX-FileCopyrightText: © 2022 ekvip automation GmbH <info@ekvip.de>
| SPDX-License-Identifier: Apache-2.0
| For details check: Apache-2.0_

.. _Apache-2.0: https://www.apache.org/licenses/LICENSE-2.0

.. </legal notes>

parameters
=================

*)

METHOD lenghtIsBetween
VAR_INPUT
	(* current string to check *)
	stringToCheck	:WSTRING(Tc2_System.MAX_STRING_LENGTH);
	(* lower limit of the string length *)
	minLenght		:USINT;
	(* upper limit of the string length *)
	maxLenght		:USINT;
	(* message if the assertion is false *)
	message			:AssertMessage;
END_VAR
THIS^.assertion.utf16LengthIsBetween(
	stringToCheck	:= ADR(stringToCheck),
	minLenght		:= minLenght,
	maxLenght		:= maxLenght,
	message			:= message
);
END_METHOD

(*

short summary
=================
This assertion method checks if the current string ``stringToCheck`` length
is equal to ``expectedLength``

.. <legal notes>

legal notes
=================
| SPDX-FileCopyrightText: © 2022 ekvip automation GmbH <info@ekvip.de>
| SPDX-License-Identifier: Apache-2.0
| For details check: Apache-2.0_

.. _Apache-2.0: https://www.apache.org/licenses/LICENSE-2.0

.. </legal notes>

parameters
=================

*)

METHOD lenghtIsExact
VAR_INPUT
	(* current string to check *)
	stringToCheck	:WSTRING(Tc2_System.MAX_STRING_LENGTH);
	(* expected length of ``stringToCheck`` *)
	expectedLength	:USINT;
	(* message if the assertion is false *)
	message			:AssertMessage;
END_VAR
THIS^.assertion.utf16LenghtIsExact(
	stringToCheck	:= ADR(stringToCheck),
	expectedLength	:= expectedLength,
	message			:= message
);
END_METHOD

(*

short summary
=================
This assertion method checks if the current string ``stringToCheck`` length
is equal or less than to ``maxLength``

.. <legal notes>

legal notes
=================
| SPDX-FileCopyrightText: © 2022 ekvip automation GmbH <info@ekvip.de>
| SPDX-License-Identifier: Apache-2.0
| For details check: Apache-2.0_

.. _Apache-2.0: https://www.apache.org/licenses/LICENSE-2.0

.. </legal notes>

parameters
=================

*)

METHOD lenghtIsMax
VAR_INPUT
	(* current string to check *)
	stringToCheck	:WSTRING(Tc2_System.MAX_STRING_LENGTH);
	(* upper limit of the length of ``stringToCheck`` *)
	maxLength		:USINT;
	(* message if the assertion is false *)
	message			:AssertMessage;
END_VAR
THIS^.assertion.utf16LenghtIsMax(
	stringToCheck	:= ADR(stringToCheck),
	maxLength		:= maxLength,
	message			:= message
);
END_METHOD

(*

short summary
=================
This assertion method checks if the current string ``stringToCheck`` length
is equal or grater than to ``minLength``

.. <legal notes>

legal notes
=================
| SPDX-FileCopyrightText: © 2022 ekvip automation GmbH <info@ekvip.de>
| SPDX-License-Identifier: Apache-2.0
| For details check: Apache-2.0_

.. _Apache-2.0: https://www.apache.org/licenses/LICENSE-2.0

.. </legal notes>

parameters
=================

*)

METHOD lenghtIsMin
VAR_INPUT
	(* current string to check *)
	stringToCheck	:WSTRING(Tc2_System.MAX_STRING_LENGTH);
	(* lower limit of the length of ``stringToCheck`` *)
	minLength		:USINT;
	(* message if the assertion is false *)
	message			:AssertMessage;
END_VAR
THIS^.assertion.utf16LenghtIsMin(
	stringToCheck	:= ADR(stringToCheck),
	minLength		:= minLength,
	message			:= message
);
END_METHOD

(*

short summary
=================
This methods is the setter for the callback class if an assertion was false

.. <legal notes>

legal notes
=================
| SPDX-FileCopyrightText: © 2022 ekvip automation GmbH <info@ekvip.de>
| SPDX-License-Identifier: Apache-2.0
| For details check: Apache-2.0_

.. _Apache-2.0: https://www.apache.org/licenses/LICENSE-2.0

.. </legal notes>

parameters
=================

*)

METHOD setCallBack
VAR_INPUT
	(* the class that must be informed if an assertion is false *)
	callBack	:IAssertCallback;  
END_VAR
SUPER^.setCallBack(callBack);
THIS^.assertion.setCallBack(callBack);
END_METHOD

(*

short summary
=================
This assertion method checks if the current string ``stringToCheck`` starts with ``start``

.. attention:: 
	start of the string is **ALWAYS** the left side of the string 
	even for writings which written from right to left like Hebrew or Arabic

.. <legal notes>

legal notes
=================
| SPDX-FileCopyrightText: © 2022 ekvip automation GmbH <info@ekvip.de>
| SPDX-License-Identifier: Apache-2.0
| For details check: Apache-2.0_

.. _Apache-2.0: https://www.apache.org/licenses/LICENSE-2.0

.. </legal notes>

parameters
=================

*)

METHOD startsWith
VAR_INPUT
	(* current string to check *)
	stringToCheck	:WSTRING(Tc2_System.MAX_STRING_LENGTH);
	(* expected start of ``stringToCheck`` *)
	start			:WSTRING(Tc2_System.MAX_STRING_LENGTH);
	(* ``TRUE`` means ignore cases; ``FALSE`` means cases must be equal too *)
	ignoreCases		:BOOL;
	(* ``TRUE`` means truncation of spaces on the left side of ``stringToCheck``*)
	trim			:BOOL;
	(* message if the assertion is false *)
	message			:AssertMessage;
END_VAR
THIS^.assertion.utf16StartsWith(
	stringToCheck	:= ADR(stringToCheck),
	start			:= ADR(start),
	ignoreCases		:= ignoreCases,
	trim			:= trim,
	message			:= message
);
END_METHOD

END_FUNCTION_BLOCK

// ---- Assertor/Assertions/StringAssertion/WString/classes/Utf16StringPointerAssertions.TcPOU
(*

short summary
=================
This class provides assert statements for UTF-16 strings

.. attention:: 
	All strings are handled as null terminated word streams.
	For UTF-16 is end of the string 16#00_00

.. <legal notes>

legal notes
=================
| SPDX-FileCopyrightText: © 2022 ekvip automation GmbH <info@ekvip.de>
| SPDX-License-Identifier: Apache-2.0
| For details check: Apache-2.0_

.. _Apache-2.0: https://www.apache.org/licenses/LICENSE-2.0

.. </legal notes>

methods and properties
=======================

*)

{attribute 'reflection'}
FUNCTION_BLOCK INTERNAL Utf16StringPointerAssertions EXTENDS AbstarctStringPointerAssertions IMPLEMENTS IUtf16StringPointerAssertions
VAR
END_VAR

(*

short summary
=================
This abstract property returns the class name of the concrete object, 
It's for debugging purpose

.. <legal notes>

legal notes
=================
| SPDX-FileCopyrightText: © 2022 ekvip automation GmbH <info@ekvip.de>
| SPDX-License-Identifier: Apache-2.0
| For details check: Apache-2.0_

.. _Apache-2.0: https://www.apache.org/licenses/LICENSE-2.0

.. </legal notes>

*)

PROPERTY className :CNM_AbstractObject.ClassName
GET
className := 'CNM_AssertionInterfaceLib.Utf16StringPointerAssertions';
END_GET
END_PROPERTY

(*

short summary
=================
this methods copy a string and returns the start address of new string

.. <legal notes>

legal notes
=================
| SPDX-FileCopyrightText: © 2022 ekvip automation GmbH <info@ekvip.de>
| SPDX-License-Identifier: Apache-2.0
| For details check: Apache-2.0_

.. _Apache-2.0: https://www.apache.org/licenses/LICENSE-2.0

.. </legal notes>

parameters
=================
:return: start address of the UTF-16 string copy

*)

METHOD PROTECTED getCopyOfUtf16String :POINTER TO WORD
VAR_INPUT
	(* string to copy *)
	stringAddress		:POINTER TO WORD;
	(* length of the string in words*)
	stringLengthInWord	:UDINT;
END_VAR
getCopyOfUtf16String := __NEW(WORD, stringLengthInWord);
IF (getCopyOfUtf16String <> 0) THEN
	Tc2_System.MEMCPY(
		destAddr := getCopyOfUtf16String,
		srcAddr := stringAddress,
		n := stringLengthInWord * SIZEOF(WORD)
	);
END_IF
END_METHOD

(*

short summary
=================
this methods copy a string and returns the start address of new string,
all small letters are capitalized in the new string.

.. <legal notes>

legal notes
=================
| SPDX-FileCopyrightText: © 2022 ekvip automation GmbH <info@ekvip.de>
| SPDX-License-Identifier: Apache-2.0
| For details check: Apache-2.0_

.. _Apache-2.0: https://www.apache.org/licenses/LICENSE-2.0

.. </legal notes>

parameters
=================
:return: start address of the UTF-16 string. 
If ``createNewUpperCaseString`` is ``TRUE`` then it's a new string

*)

METHOD PROTECTED getNewUtf16UCaseString :POINTER TO WORD; 
VAR_INPUT
	(* start address of the string to copy and capitalize *)
	stringAddress				:POINTER TO WORD;
	(* length of the string ``stringAddress`` *)
	stringLengthInWord			:UDINT;
	(* 
	``TRUE means meake a copy and capitalize it, 
	``FALSE`` means return just ``stringAddress``
	and do nothing else
	*)
	createNewUpperCaseString	:BOOL;
END_VAR
IF (createNewUpperCaseString) THEN
	getNewUtf16UCaseString := THIS^.getCopyOfUtf16String(stringAddress, stringLengthInWord);
	THIS^.utf16UpperCase(getNewUtf16UCaseString, stringLengthInWord);
ELSE
	getNewUtf16UCaseString := stringAddress;
END_IF
END_METHOD

(*

short summary
=================
This methods returns the length of a null terminated UTF-16 string.
The returned length is in characters (in UTF-16 have some charcters 32 bit length).
This method provides two outputs to get the length in byte and word, too. 

.. attention:: 
	All strings are handled as null terminated byte streams.
	For UTF-16 is end of the string 16#00_00

.. <legal notes>

legal notes
=================
| SPDX-FileCopyrightText: © 2022 ekvip automation GmbH <info@ekvip.de>
| SPDX-License-Identifier: Apache-2.0
| For details check: Apache-2.0_

.. _Apache-2.0: https://www.apache.org/licenses/LICENSE-2.0

.. </legal notes>

parameters
=================
:return: length of the UTF-16 string in characters

*)

METHOD PROTECTED getUtf16StringLength :UDINT
VAR_INPUT
	(* Start address of the string for which the length is to be determined *)
	stringAddress	:POINTER TO WORD;
END_VAR
VAR_OUTPUT
	(* sting length in bytes *)
	lengthInByte	:UDINT;
	(* string length in words *)
	lengthInWord	:UDINT;
END_VAR
VAR
	(* character index to iterate thru the string *)
	character		:UDINT;
END_VAR
VAR CONSTANT
	(* NUL it terminates the string *)
	END_OF_STRING		:WORD := 16#0000;
	(* byte counter *)
	INCREMENT_LENGTH	:UDINT := 1;
END_VAR
getUtf16StringLength	:= 0;
lengthInByte		:= 0;
character			:= 0; 
lengthInWord		:= 0;

IF (stringAddress = 0) THEN
	RETURN;
END_IF

WHILE (stringAddress[character] <> END_OF_STRING) DO
	getUtf16StringLength := getUtf16StringLength + 1;
	IF (THIS^.isUtf16CharASurrogatePair(
			highWord := stringAddress[character], 
			lowWord := stringAddress[character+1]
		)
	) THEN
		character := character + 2;
		lengthInByte := lengthInByte + 4;
	ELSE
		character := character + 1;
		lengthInByte := lengthInByte + 2;		
	END_IF;
END_WHILE

//add one word for null termination, it's required for the surrogate pair check
lengthInWord := character + 1;
lengthInByte := lengthInByte + 2;
END_METHOD

(*

short summary
=================
This methods calculates from an UTF-32 code-point_ an UTF-16 surrogate-pair_

.. _surrogate-pair: https://en.wikipedia.org/wiki/UTF-16#U+D800_to_U+DFFF

.. _code-point: https://en.wikipedia.org/wiki/UTF-16#Code_points_from_U+010000_to_U+10FFFF

.. <legal notes>

legal notes
=================
| SPDX-FileCopyrightText: © 2022 ekvip automation GmbH <info@ekvip.de>
| SPDX-License-Identifier: Apache-2.0
| For details check: Apache-2.0_

.. _Apache-2.0: https://www.apache.org/licenses/LICENSE-2.0

.. </legal notes>

parameters
=================

*)

METHOD PROTECTED getUtf16SurrogatePairFromUtf32
VAR_INPUT
	(* utf32 code point *)
	utf32Char	:DWORD;
END_VAR
VAR_OUTPUT
	(* high word of the surrogate pair *)
	highWord	:WORD;
	(* low word of the surrogate pair *)
	lowWord		:WORD;
END_VAR
utf32Char := utf32Char - 16#10000;
highWord := TO_WORD(SHR(utf32Char, 10)) + 16#D800;
lowWord	:= TO_WORD(utf32Char AND 16#3FF) + 16#DC00;
END_METHOD

(*

short summary
=================
This methods calculates from an UTF-16 surrogate-pair_ an UTF-32 code-point_

.. _surrogate-pair: https://en.wikipedia.org/wiki/UTF-16#U+D800_to_U+DFFF

.. _code-point: https://en.wikipedia.org/wiki/UTF-16#Code_points_from_U+010000_to_U+10FFFF

.. <legal notes>

legal notes
=================
| SPDX-FileCopyrightText: © 2022 ekvip automation GmbH <info@ekvip.de>
| SPDX-License-Identifier: Apache-2.0
| For details check: Apache-2.0_

.. _Apache-2.0: https://www.apache.org/licenses/LICENSE-2.0

.. </legal notes>

parameters
=================
:return: UTF-32 character (code-point) from the UTF-16 surrogate pair

*)

METHOD PROTECTED getUtf32FromUtf16SurrogatePair :DWORD
VAR_INPUT
	(* high word of the surrogate pair *)
	highWord	:WORD;
	(* low word of the surrogate pair *)
	lowWord		:WORD;
END_VAR
getUtf32FromUtf16SurrogatePair := ((
		SHL(TO_DWORD(highWord - 16#D800), 10)
	) + (
		(TO_DWORD(lowWord - 16#DC00) + 16#10000)
	)
);
END_METHOD

(*

short summary
=================
this methods checks if an UTF-16 character is a whitespace character

.. <legal notes>

legal notes
=================
| SPDX-FileCopyrightText: © 2022 ekvip automation GmbH <info@ekvip.de>
| SPDX-License-Identifier: Apache-2.0
| For details check: Apache-2.0_

.. _Apache-2.0: https://www.apache.org/licenses/LICENSE-2.0

.. </legal notes>

parameters
=================
:return: ``TRUE`` means ``character`` is whitespace,
``FALSE`` means ``character`` is no whitespace 

*)

METHOD PROTECTED isCharUtf16WhiteSpace :BOOL
VAR_INPUT
	(* character to check if it's whitespace *)
	character	:WORD;
END_VAR
VAR CONSTANT
	HORIZONTAL_TAB				:WORD := 16#0009;
	LINE_FEED					:WORD := 16#000A;
	VERTICAL_TAB				:WORD := 16#000B;
	FROM_FEED					:WORD := 16#000C;
	CARRIAGE_RETURN				:WORD := 16#000D;
	SPACE						:WORD := 16#0020;
	NEXT_LINE					:WORD := 16#0085;
	NO_BREAK_SPACE				:WORD := 16#00A0;
	OGHAM_SPACE_MARK			:WORD := 16#1680;
	EN_QUAD						:WORD := 16#2000;
	EM_QUAD						:WORD := 16#2001;
	EN_SPACE					:WORD := 16#2002;
	EM_SPACE					:WORD := 16#2003;
	THREE_PER_EM_SPACE			:WORD := 16#2004;
	FOUR_PER_EM_SPACE			:WORD := 16#2005;
	SIX_PER_EM_SPACE			:WORD := 16#2006;
	FIGURE_SPACE				:WORD := 16#2007;
	PUNCTUATION_SPACE			:WORD := 16#2008;
	THIN_SPACE					:WORD := 16#2009;
	HAIR_SPACE					:WORD := 16#200A;
	LINE_SEPERATOR				:WORD := 16#2028;
	PARAGRAPH_SEPERATOR 		:WORD := 16#2029;
	NARROW_NO_BREAK_SPACE		:WORD := 16#202F;
	MEDIUM_MATHEMEATICAL_SPACE	:WORD := 16#205F;
	IDEOGRAPHIC_SPACE			:WORD := 16#3000;
END_VAR
CASE character OF
HORIZONTAL_TAB .. CARRIAGE_RETURN,
SPACE,
NEXT_LINE,
NO_BREAK_SPACE,
OGHAM_SPACE_MARK,
EN_QUAD .. HAIR_SPACE,
LINE_SEPERATOR .. PARAGRAPH_SEPERATOR,
MEDIUM_MATHEMEATICAL_SPACE,
IDEOGRAPHIC_SPACE:
	isCharUtf16WhiteSpace := TRUE;
ELSE
	isCharUtf16WhiteSpace := FALSE;	
END_CASE
END_METHOD

(*

short summary
=================
This methods checks if two UTF-16 characters are a surrogate-pair_

.. _surrogate-pair: https://en.wikipedia.org/wiki/UTF-16#U+D800_to_U+DFFF

.. <legal notes>

legal notes
=================
| SPDX-FileCopyrightText: © 2022 ekvip automation GmbH <info@ekvip.de>
| SPDX-License-Identifier: Apache-2.0
| For details check: Apache-2.0_

.. _Apache-2.0: https://www.apache.org/licenses/LICENSE-2.0

.. </legal notes>

parameters
=================
:return: ``TRUE`` means it's a surrogate pair,
``FALSE`` means it's no surrogate pair

*)

METHOD PROTECTED isUtf16CharASurrogatePair :BOOL
VAR_INPUT
	(* high word of the surrogate pair *)
	highWord	:WORD;
	(* low word of the surrogate pair *)
	lowWord		:WORD;
END_VAR
isUtf16CharASurrogatePair := (
	(highWord >= 16#D800)
	AND (highWord <= 16#DBFF)
	AND (lowWord >= 16#DC00)
	AND (lowWord <= 16#DFFF)
);
END_METHOD

(*

short summary
=================
This method converts an UTF-16 lowercase character to an UTF-16 uppercase character.

.. <legal notes>

legal notes
=================
| SPDX-FileCopyrightText: © 2022 ekvip automation GmbH <info@ekvip.de>
| SPDX-License-Identifier: Apache-2.0
| For details check: Apache-2.0_

.. _Apache-2.0: https://www.apache.org/licenses/LICENSE-2.0

.. </legal notes>

parameters
=================

*)

METHOD PROTECTED upperCaseUtf16Char
VAR_IN_OUT
	(* utf-16 char to upper case *)
	char		:WORD;
END_VAR
CASE char OF
16#0061 .. 16#007A,
16#00E0 .. 16#00F6,
16#00F8 .. 16#00FE,
16#03B1 .. 16#03C1,
16#03C3 .. 16#03CB,
16#0430 .. 16#044F,
16#FF41 .. 16#FF5A:
	char := char - 16#0020;
16#00B5:
	char := 16#039C;
16#00DF,
16#017F:
	char := 16#0053;
16#00FF:
	char := 16#0178;
16#0101 .. 16#012F,
16#0132 .. 16#0137,
16#013A .. 16#0148,
16#014B .. 16#0177,
16#017A .. 16#017E,
16#0183 .. 16#0185,
16#0188,
16#018C,
16#0192,
16#0199,
16#01A1 .. 16#01A5,
16#01A8,
16#01AD,
16#01B0,
16#01B4,
16#01B6,
16#01B9,
16#01BD,
16#01CE .. 16#01DC,
16#01DF,
16#01E1 .. 16#01EF,
16#01F5,
16#01FB .. 16#0217,
16#03E3 .. 16#03EF,
16#0461 .. 16#0481,
16#0491 .. 16#04BF,
16#04C2 .. 16#04C4,
16#04C8,
16#04CC,
16#04D1 .. 16#04EB,
16#04EF .. 16#04F5,
16#04F9,
16#1E01 .. 16#1E95,
16#1EA1 .. 16#1EF9:
	char := SEL((char.0 = 1), char, (char := char-1));
16#0131:
	char := 16#0049;
16#0180:
	char := 16#0243;
16#01C6,
16#01C9,
16#01CC,
16#01F3:
	char := SEL((char.0 = 0), char, (char := char-2));
16#0253:
	char := 16#0181;
16#0254:
	char := 16#0186;
16#0257,
16#0260:
	char := char - 16#00CD;
16#0258,
16#0259:
	char := char - 16#00CA;
16#025B:
	char := 16#0190;
16#0263:
	char := 16#0194;
16#0268:
	char := 16#0197;
16#0269,
16#026F:
	char := char - 16#00D3;
16#0276:
	char := 16#019D;
16#0275:
	char := 16#019F;
16#0283,
16#0288:
	char := char - 16#00DA;
16#028A .. 16#028B:
	char := char - 16#00D9;
16#0292:
	char := 16#01B7;
16#03AC:
	char := 16#0386;
16#03AD .. 16#03AF:
	char := char - 16#0025;
16#03CC:
	char := 16#038C;
16#03CD .. 16#03CE:
	char := char - 16#003F;
16#0451 .. 16#045C,
16#045E .. 16#045F:
	char := char - 16#0050;
16#0561 .. 16#0586,
16#10D0 .. 16#10F5:		
	char := char - 16#0030;
16#1F00 .. 16#1F07,
16#1F10 .. 16#1F15,
16#1F20 .. 16#1F27,
16#1F30 .. 16#1F37,
16#1F40 .. 16#1F45,
16#1F51,
16#1F53,
16#1F55,
16#1F57,
16#1F60 .. 16#1F67,
16#1F80 .. 16#1F87,
16#1F90 .. 16#1F97,
16#1FA0 .. 16#1FA7,
16#1FB0 .. 16#1FB1,
16#1FD0 .. 16#1FD1,
16#1FE0 .. 16#1FE1:
	char := char + 16#0008;
16#24D0 .. 16#24E9:		
	char := char - 16#001A;
ELSE
	RETURN;
END_CASE
END_METHOD

(*

short summary
=================
This method converts an UTF-32 lowercase character to an UTF-32 uppercase character.

.. <legal notes>

legal notes
=================
| SPDX-FileCopyrightText: © 2022 ekvip automation GmbH <info@ekvip.de>
| SPDX-License-Identifier: Apache-2.0
| For details check: Apache-2.0_

.. _Apache-2.0: https://www.apache.org/licenses/LICENSE-2.0

.. </legal notes>

parameters
=================

*)

METHOD PROTECTED upperCaseUtf32Char
VAR_IN_OUT
	(* utf-32 char to upper case *)
	char		:DWORD;
END_VAR
CASE char OF
16#00010428 .. 16#00010447,
16#000104D8 .. 16#000104FB:
	char := char - 16#00000028;
16#00010CC0 .. 16#00010CF2:
	char := char - 16#00000040;
16#000118C0 .. 16#000118DF,
16#00016E60 .. 16#00016E7F:
	char := char - 16#00000020;
16#0001D41A .. 16#0001D433,
16#0001D44E .. 16#0001D454,
16#0001D456 .. 16#0001D467,
16#0001D482 .. 16#0001D49B,
16#0001D4B6,
16#0001D4B8 .. 16#0001D4B9,
16#0001D4BF .. 16#0001D4C0,
16#0001D4C3,
16#0001D4C5 .. 16#0001D4C6,
16#0001D4C8 .. 16#0001D4CF,
16#0001D4EA .. 16#0001D503,
16#0001D51E .. 16#0001D51F,
16#0001D521 .. 16#0001D524,
16#0001D527 .. 16#0001D52E,
16#0001D530 .. 16#0001D536,
16#0001D552 .. 16#0001D553,
16#0001D555 .. 16#0001D558,
16#0001D55A .. 16#0001D55E,
16#0001D560,
16#0001D564 .. 16#0001D56A,
16#0001D586 .. 16#0001D59F,
16#0001D5BA .. 16#0001D5D3,
16#0001D5EE .. 16#0001D607,
16#0001D622 .. 16#0001D63B,
16#0001D656 .. 16#0001D66F,
16#0001D68A .. 16#0001D6A3,
16#0001D6C2 .. 16#0001D6E1,
16#0001D6FC .. 16#0001D71B,
16#0001D736 .. 16#0001D755,
16#0001D770 .. 16#0001D78F,
16#0001D7AA .. 16#0001D7C9:
	char := char - 16#0000001A;
16#0001D7CB:
	char := 16#0001D7CA;
16#0001E922 .. 16#0001E943:
	char := char - 16#00000022;
ELSE
	RETURN;
END_CASE
END_METHOD

(*

short summary
=================
This methods checks if the high word an UTF-16 surrogate-pair_
is inside the range of characters with lower and upper case

.. _surrogate-pair: https://en.wikipedia.org/wiki/UTF-16#U+D800_to_U+DFFF

.. <legal notes>

legal notes
=================
| SPDX-FileCopyrightText: © 2022 ekvip automation GmbH <info@ekvip.de>
| SPDX-License-Identifier: Apache-2.0
| For details check: Apache-2.0_

.. _Apache-2.0: https://www.apache.org/licenses/LICENSE-2.0

.. </legal notes>

parameters
=================
:return: ``TRUE`` means it could be letter with lower and uppercase,
``FALSE`` means this is no letter with lower and upper case

*)

METHOD PROTECTED utf16CharIsSurrogateHighWordLetterLike :BOOL
VAR_IN_OUT
	highWord	:WORD;
END_VAR
utf16CharIsSurrogateHighWordLetterLike := FALSE;
CASE highWord OF
16#D801,
16#D803,
16#D806,
16#D81B,
16#D835,
16#D83A:
	utf16CharIsSurrogateHighWordLetterLike := TRUE;
ELSE
	RETURN;
END_CASE
END_METHOD

(*

short summary
=================
This assertion method for UTF-16 strings checks if the current string ``stringToCheck`` contains the search string ``searchString``

.. attention:: 
	All strings are handled as null terminated word streams.
	For UTF-16 is end of the string 16#00_00

.. <legal notes>

